  MoveL 686 to (-94.83, -177.34, 370.15) mm, rotated rx -20.04 ry 0.01 rz 0 deg; joints [12.615, -131.611, -68.908, -59.593, 88.727, 7.17]
  MoveL 687 to (-95.13, -172.76, 368.52) mm, rotated rx -19.93 ry 0.38 rz -0.14 deg; joints [12.853, -130.937, -70.265, -58.86, 88.278, 7.403]
  MoveL 688 to (-95.18, -165.44, 365.46) mm, rotated rx -20.3 ry 0.73 rz -0.27 deg; joints [13.07, -130.12, -71.703, -58.656, 87.921, 7.628]
  MoveL 689 to (-94.96, -155.27, 361.72) mm, rotated rx -19.76 ry 0.12 rz -0.04 deg; joints [12.925, -128.559, -74.952, -56.346, 88.521, 7.469]
  MoveL 690 to (-95.06, -148.96, 360) mm, rotated rx -19.41 ry -0.34 rz 0.12 deg; joints [12.816, -127.682, -76.899, -54.857, 88.972, 7.352]
  MoveL 691 to (-89.88, -148.96, 360) mm, rotated rx -19.07 ry -0.33 rz 0.11 deg; joints [12.421, -127.542, -77.28, -54.28, 88.998, 6.956]
  MoveL 692 to (-94.67, -143.58, 357.81) mm, rotated rx -19.21 ry -0.64 rz 0.22 deg; joints [12.719, -126.92, -78.436, -53.844, 89.284, 7.251]
  MoveL 693 to (-95.24, -134.75, 355.85) mm, rotated rx -19.89 ry -0.83 rz 0.3 deg; joints [12.73, -126.323, -79.629, -53.895, 89.571, 7.278]
  MoveL 694 to (-95.24, -124.99, 352.14) mm, rotated rx -20.45 ry -1.05 rz 0.39 deg; joints [12.704, -125.412, -81.243, -53.713, 89.885, 7.264]
  MoveL 695 to (-92.42, -119.21, 350) mm, rotated rx -20.35 ry -1.23 rz 0.46 deg; joints [12.457, -124.708, -82.656, -52.889, 90.101, 7.019]
  MoveL 696 to (-95.21, -114.33, 347.08) mm, rotated rx -20.45 ry -1.17 rz 0.44 deg; joints [12.774, -124.04, -83.727, -52.59, 89.995, 7.334]
  MoveL 697 to (-95.11, -104.56, 343.32) mm, rotated rx -20.25 ry -1.28 rz 0.47 deg; joints [12.838, -122.816, -86.139, -51.19, 90.078, 7.393]
  MoveL 698 to (-95.03, -94.94, 340.98) mm, rotated rx -19.38 ry -1.18 rz 0.41 deg; joints [13.046, -121.51, -89.146, -48.641, 89.811, 7.577]
  MoveL 699 to (-91.55, -89.14, 340) mm, rotated rx -19.07 ry -1.15 rz 0.4 deg; joints [12.839, -120.897, -90.647, -47.446, 89.781, 7.365]
  MoveL 700 to (-95.44, -84.4, 336.73) mm, rotated rx -19.11 ry -1.33 rz 0.46 deg; joints [13.163, -120.206, -91.7, -47.101, 89.907, 7.684]
  MoveL 701 to (-95.05, -75.22, 333) mm, rotated rx -20.06 ry -1.49 rz 0.54 deg; joints [13.102, -119.543, -92.613, -47.764, 90.223, 7.648]
  MoveL 702 to (-95.12, -66.84, 330.77) mm, rotated rx -20.48 ry -1.53 rz 0.57 deg; joints [13.159, -118.908, -93.858, -47.567, 90.322, 7.714]
  MoveL 703 to (-95.11, -61.19, 328.48) mm, rotated rx -20.08 ry -1.43 rz 0.52 deg; joints [13.317, -118.116, -95.454, -46.38, 90.126, 7.86]
  MoveL 704 to (-94.95, -54.68, 325.45) mm, rotated rx -20.03 ry -1.3 rz 0.47 deg; joints [13.468, -117.321, -96.854, -45.745, 89.952, 8.008]
  MoveL 705 to (-95.13, -44.85, 322.06) mm, rotated rx -19.59 ry -1.28 rz 0.45 deg; joints [13.666, -116.156, -99.258, -44.08, 89.831, 8.191]
  MoveL 706 to (-93.28, -38.74, 320) mm, rotated rx -19.37 ry -1.41 rz 0.49 deg; joints [13.524, -115.48, -100.669, -43.099, 89.961, 8.045]
  MoveL 707 to (-95.27, -34.68, 317.51) mm, rotated rx -19.05 ry -1.44 rz 0.5 deg; joints [13.789, -114.821, -101.831, -42.28, 89.901, 8.297]
  MoveL 708 to (-95, -25.83, 315.53) mm, rotated rx -19.14 ry -1.47 rz 0.51 deg; joints [13.868, -114.108, -103.402, -41.504, 89.923, 8.377]
  MoveL 709 to (-95.26, -15.36, 311.91) mm, rotated rx -18.64 ry -1.49 rz 0.5 deg; joints [14.085, -112.917, -105.883, -39.713, 89.831, 8.575]
  MoveL 710 to (-94.57, -9.01, 310) mm, rotated rx -18.16 ry -1.4 rz 0.46 deg; joints [14.208, -112.189, -107.516, -38.36, 89.638, 8.681]
  MoveL 711 to (-94.8, -3.67, 307.71) mm, rotated rx -17.94 ry -1.19 rz 0.39 deg; joints [14.466, -111.532, -108.75, -37.596, 89.329, 8.926]
  MoveL 712 to (-94.93, 5.41, 304.51) mm, rotated rx -17.3 ry -1.12 rz 0.35 deg; joints [14.744, -110.468, -111.026, -35.775, 89.086, 9.176]
  MoveL 713 to (-95.04, 14.85, 302.51) mm, rotated rx -17.21 ry -1.01 rz 0.31 deg; joints [14.992, -109.714, -112.788, -34.694, 88.907, 9.414]
  MoveL 714 to (-94.95, 23.14, 300.98) mm, rotated rx -17.62 ry -1.13 rz 0.36 deg; joints [15.02, -109.237, -113.848, -34.497, 89.087, 9.457]
  MoveL 715 to (-95.55, 28.29, 298.3) mm, rotated rx -18.2 ry -1.07 rz 0.35 deg; joints [15.17, -108.771, -114.269, -35.132, 89.097, 9.625]
  MoveL 716 to (-95.03, 35.17, 294.87) mm, rotated rx -19.11 ry -0.94 rz 0.33 deg; joints [15.247, -108.211, -114.702, -36.172, 89.104, 9.73]
  MoveL 717 to (-94.91, 45.46, 291.79) mm, rotated rx -19.49 ry -1.08 rz 0.38 deg; joints [15.308, -107.423, -116.156, -35.863, 89.307, 9.803]
  MoveL 718 to (-93.25, 51.3, 290) mm, rotated rx -18.82 ry -1.28 rz 0.44 deg; joints [15.184, -106.745, -117.783, -34.216, 89.42, 9.659]
  MoveL 719 to (-95.13, 55.87, 287.9) mm, rotated rx -18.18 ry -1.04 rz 0.34 deg; joints [15.727, -106.043, -119.212, -32.903, 88.951, 10.169]
  MoveL 720 to (-95.02, 65.32, 284.92) mm, rotated rx -17.88 ry -0.65 rz 0.21 deg; joints [16.219, -105.1, -121.129, -31.723, 88.389, 10.641]
  MoveL 721 to (-94.97, 75, 282.29) mm, rotated rx -17.01 ry -0.47 rz 0.14 deg; joints [16.669, -104.106, -123.55, -29.499, 87.945, 11.045]
  MoveL 722 to (-95.57, 81.71, 280.31) mm, rotated rx -16.74 ry -0.5 rz 0.15 deg; joints [16.933, -103.484, -124.933, -28.476, 87.854, 11.29]
  MoveL 723 to (-94.86, 86.85, 278.18) mm, rotated rx -16.68 ry -0.56 rz 0.17 deg; joints [16.947, -102.95, -125.872, -27.996, 87.91, 11.3]
  MoveL 724 to (-95.16, 94.95, 276.16) mm, rotated rx -16.91 ry -0.57 rz 0.17 deg; joints [17.159, -102.378, -127.022, -27.649, 87.916, 11.518]
  MoveL 725 to (-96.68, 102.58, 275.65) mm, rotated rx -15.92 ry -0.81 rz 0.23 deg; joints [17.522, -101.885, -129.109, -25.048, 87.866, 11.821]
  MoveL 726 to (-84.81, -254.16, 398.04) mm, rotated rx -18.14 ry -0.49 rz 0.16 deg; joints [11.089, -142.234, -48.176, -67.726, 89.323, 5.629]
  MoveL 727 to (-84.83, -246.42, 397.43) mm, rotated rx -19.51 ry -0.51 rz 0.18 deg; joints [11.08, -142.169, -48.262, -69.063, 89.483, 5.647]
  MoveL 728 to (-84.96, -235.69, 393.28) mm, rotated rx -20.66 ry -0.69 rz 0.26 deg; joints [11.053, -141.138, -50.022, -69.462, 89.799, 5.64]
  MoveL 729 to (-84.27, -228.62, 390.27) mm, rotated rx -20.97 ry -1.13 rz 0.43 deg; joints [10.868, -140.127, -51.941, -68.816, 90.332, 5.462]
  MoveL 730 to (-85.04, -223.33, 387.97) mm, rotated rx -21.99 ry -1.35 rz 0.55 deg; joints [10.834, -139.957, -52.001, -69.91, 90.674, 5.445]
  MoveL 731 to (-84.87, -214.7, 385.26) mm, rotated rx -22.47 ry -1.84 rz 0.76 deg; joints [10.661, -138.951, -54.007, -69.339, 91.279, 5.28]
  MoveL 732 to (-84.93, -206.09, 382.19) mm, rotated rx -22.25 ry -2.23 rz 0.91 deg; joints [10.573, -137.441, -57.118, -67.482, 91.687, 5.191]
  MoveL 733 to (-85.21, -200.4, 379) mm, rotated rx -21.97 ry -2.25 rz 0.91 deg; joints [10.642, -136.244, -59.41, -66.099, 91.667, 5.255]
  MoveL 734 to (-84.67, -194.51, 376.22) mm, rotated rx -21.82 ry -2.22 rz 0.89 deg; joints [10.665, -135.201, -61.427, -64.985, 91.616, 5.276]
  MoveL 735 to (-85.3, -184.88, 372.55) mm, rotated rx -21.44 ry -1.6 rz 0.63 deg; joints [11.069, -133.516, -64.805, -62.969, 90.844, 5.669]
  MoveL 736 to (-85.21, -177.44, 370.35) mm, rotated rx -20.98 ry -0.87 rz 0.33 deg; joints [11.454, -132.242, -67.486, -61.195, 89.957, 6.042]
  MoveL 737 to (-85.03, -172.64, 368.48) mm, rotated rx -20.75 ry -0.44 rz 0.17 deg; joints [11.679, -131.432, -69.11, -60.203, 89.44, 6.26]
  MoveL 738 to (-84.94, -165.44, 365.46) mm, rotated rx -20.37 ry -0.12 rz 0.04 deg; joints [11.9, -130.218, -71.536, -58.653, 89.017, 6.471]
  MoveL 739 to (-85.48, -155.44, 361.28) mm, rotated rx -19.25 ry -0.04 rz 0.01 deg; joints [12.13, -128.312, -75.522, -55.479, 88.766, 6.675]
  MoveL 740 to (-82.13, -150.42, 359) mm, rotated rx -18.73 ry -0.38 rz 0.13 deg; joints [11.782, -127.423, -77.38, -53.941, 89.136, 6.321]
  MoveL 741 to (-84.91, -144.97, 357.61) mm, rotated rx -18.63 ry -0.52 rz 0.18 deg; joints [12.002, -126.775, -78.786, -53.071, 89.225, 6.534]
  MoveL 742 to (-85.11, -135.15, 355.64) mm, rotated rx -19.31 ry -0.98 rz 0.34 deg; joints [11.863, -126.118, -80.166, -52.971, 89.812, 6.412]
  MoveL 743 to (-84.89, -125.22, 352.31) mm, rotated rx -20.49 ry -1.36 rz 0.51 deg; joints [11.702, -125.532, -81.043, -53.799, 90.384, 6.278]
  MoveL 744 to (-81.66, -120.69, 349) mm, rotated rx -21 ry -1.04 rz 0.4 deg; joints [11.61, -125.044, -81.552, -54.323, 90.118, 6.196]
  MoveL 745 to (-87.84, -119.21, 350) mm, rotated rx -20.58 ry -1.12 rz 0.42 deg; joints [12.117, -124.823, -82.364, -53.302, 90.066, 6.689]
  MoveL 746 to (-84.74, -114.13, 347.26) mm, rotated rx -20.77 ry -0.68 rz 0.26 deg; joints [12.109, -124.213, -83.322, -53.205, 89.633, 6.684]
  MoveL 747 to (-84.88, -104.45, 343.56) mm, rotated rx -19.91 ry -0.89 rz 0.32 deg; joints [12.172, -122.715, -86.477, -50.661, 89.737, 6.729]
  MoveL 748 to (-85.9, -95.32, 340.81) mm, rotated rx -19.48 ry -1.14 rz 0.4 deg; joints [12.262, -121.594, -88.906, -48.897, 89.928, 6.808]
  MoveL 749 to (-81.76, -91.98, 339) mm, rotated rx -19.35 ry -0.99 rz 0.35 deg; joints [12.018, -121.119, -89.755, -48.418, 89.804, 6.566]
  MoveL 750 to (-87.55, -89.14, 340) mm, rotated rx -19.04 ry -1.05 rz 0.36 deg; joints [12.537, -120.9, -90.648, -47.429, 89.732, 7.068]
  MoveL 751 to (-84.71, -84.61, 337.65) mm, rotated rx -18.99 ry -0.91 rz 0.31 deg; joints [12.417, -120.311, -91.674, -46.96, 89.595, 6.95]
  MoveL 752 to (-84.95, -75.08, 332.91) mm, rotated rx -19.86 ry -1.04 rz 0.37 deg; joints [12.44, -119.469, -92.789, -47.532, 89.836, 6.991]
  MoveL 753 to (-84.91, -66.88, 330.61) mm, rotated rx -20.34 ry -1.25 rz 0.46 deg; joints [12.388, -118.87, -93.932, -47.437, 90.136, 6.951]
  MoveL 754 to (-85.07, -61.26, 328.67) mm, rotated rx -20.11 ry -1.4 rz 0.51 deg; joints [12.408, -118.2, -95.324, -46.46, 90.256, 6.966]
  MoveL 755 to (-85.02, -54.81, 325.82) mm, rotated rx -20 ry -1.41 rz 0.51 deg; joints [12.487, -117.418, -96.765, -45.692, 90.238, 7.041]
  MoveL 756 to (-84.99, -44.93, 322.16) mm, rotated rx -19.53 ry -1.38 rz 0.49 deg; joints [12.653, -116.206, -99.224, -43.982, 90.116, 7.194]
  MoveL 757 to (-83.93, -37.55, 320.41) mm, rotated rx -19.24 ry -1.48 rz 0.52 deg; joints [12.61, -115.476, -100.91, -42.732, 90.187, 7.144]
  MoveL 758 to (-85.47, -33.08, 317.84) mm, rotated rx -19.11 ry -1.45 rz 0.5 deg; joints [12.846, -114.844, -101.966, -42.181, 90.096, 7.373]
  MoveL 759 to (-85.27, -25.33, 315.56) mm, rotated rx -19.07 ry -1.36 rz 0.47 deg; joints [12.978, -114.107, -103.479, -41.378, 89.976, 7.502]
  MoveL 760 to (-84.89, -15.77, 311.74) mm, rotated rx -18.78 ry -1.43 rz 0.49 deg; joints [13.062, -113.012, -105.595, -40.06, 89.988, 7.577]
  MoveL 761 to (-85.09, -9.98, 310) mm, rotated rx -18.54 ry -1.27 rz 0.42 deg; joints [13.276, -112.393, -106.913, -39.149, 89.74, 7.78]
  MoveL 762 to (-84.8, -4.2, 307.93) mm, rotated rx -18.18 ry -1.05 rz 0.35 deg; joints [13.484, -111.701, -108.347, -38.08, 89.423, 7.974]
  MoveL 763 to (-85.06, 5.28, 305.8) mm, rotated rx -17.23 ry -0.91 rz 0.28 deg; joints [13.814, -110.671, -110.953, -35.594, 89.068, 8.266]
  MoveL 764 to (-84.99, 14.63, 301.76) mm, rotated rx -17.22 ry -1.15 rz 0.36 deg; joints [13.828, -109.688, -112.682, -34.803, 89.309, 8.279]
  MoveL 765 to (-85.77, 22.24, 300.18) mm, rotated rx -17.6 ry -1.07 rz 0.34 deg; joints [14.047, -109.203, -113.681, -34.672, 89.237, 8.506]
  MoveL 766 to (-84.15, 26.99, 298.69) mm, rotated rx -18.27 ry -1 rz 0.33 deg; joints [13.935, -108.96, -113.894, -35.376, 89.288, 8.417]
  MoveL 767 to (-85.02, 35.35, 295.86) mm, rotated rx -18.92 ry -1.06 rz 0.36 deg; joints [14.081, -108.355, -114.793, -35.714, 89.42, 8.58]
  MoveL 768 to (-85, 45.69, 292.45) mm, rotated rx -19.11 ry -1.58 rz 0.55 deg; joints [13.917, -107.501, -116.427, -35.041, 90.025, 8.424]
  MoveL 769 to (-84.93, 51.88, 290) mm, rotated rx -18.91 ry -1.75 rz 0.6 deg; joints [13.931, -106.837, -117.708, -34.199, 90.171, 8.432]
  MoveL 770 to (-85.15, 56.65, 288) mm, rotated rx -18.6 ry -1.62 rz 0.55 deg; joints [14.16, -106.243, -118.85, -33.365, 89.943, 8.648]
  MoveL 771 to (-85.04, 65.47, 285.53) mm, rotated rx -18.18 ry -1.37 rz 0.45 deg; joints [14.519, -105.381, -120.759, -31.946, 89.541, 8.986]
  MoveL 772 to (-85.04, 75.21, 282.85) mm, rotated rx -17.29 ry -1.1 rz 0.34 deg; joints [14.99, -104.363, -123.22, -29.684, 89.016, 9.415]
  MoveL 773 to (-85.08, 80.94, 280) mm, rotated rx -16.76 ry -0.95 rz 0.29 deg; joints [15.294, -103.572, -124.713, -28.488, 88.702, 9.692]
  MoveL 774 to (-84.92, 86.24, 278.23) mm, rotated rx -16.55 ry -0.92 rz 0.27 deg; joints [15.443, -103.052, -125.802, -27.719, 88.597, 9.828]
  MoveL 775 to (-84.97, 94.98, 276.23) mm, rotated rx -16.7 ry -0.91 rz 0.27 deg; joints [15.634, -102.45, -127.114, -27.169, 88.572, 10.021]
  MoveL 776 to (-85.97, 101.04, 275.32) mm, rotated rx -15.86 ry -0.92 rz 0.26 deg; joints [16.001, -101.951, -128.843, -25.117, 88.344, 10.341]
  MoveL 777 to (-73.01, -256.67, 400.33) mm, rotated rx -16.93 ry -1.96 rz 0.6 deg; joints [9.707, -142.108, -49.069, -65.622, 91.046, 4.257]
  MoveL 778 to (-76.07, -253.64, 398.85) mm, rotated rx -17.91 ry -1.49 rz 0.48 deg; joints [10.094, -142.199, -48.515, -67.094, 90.552, 4.652]
  MoveL 779 to (-74.72, -245.59, 396.62) mm, rotated rx -19.49 ry -1.5 rz 0.53 deg; joints [9.986, -142.077, -48.436, -68.867, 90.733, 4.572]
  MoveL 780 to (-75.3, -235.91, 394.03) mm, rotated rx -20.25 ry -1.47 rz 0.54 deg; joints [10.071, -141.051, -50.447, -68.643, 90.751, 4.666]
  MoveL 781 to (-74.37, -228.01, 391.14) mm, rotated rx -20.89 ry -1.46 rz 0.56 deg; joints [10.035, -140.182, -52.039, -68.557, 90.806, 4.64]
  MoveL 782 to (-75.54, -222.35, 388.11) mm, rotated rx -21.63 ry -1.6 rz 0.64 deg; joints [10.073, -139.664, -52.77, -69.061, 91.019, 4.687]
  MoveL 783 to (-74.76, -215.31, 386) mm, rotated rx -21.85 ry -2.02 rz 0.81 deg; joints [9.881, -138.752, -54.644, -68.29, 91.514, 4.5]
  MoveL 784 to (-75.09, -205.73, 383.37) mm, rotated rx -22.06 ry -2.43 rz 0.98 deg; joints [9.784, -137.492, -57.28, -67.082, 91.984, 4.408]
  MoveL 785 to (-72.03, -198.94, 380) mm, rotated rx -21.9 ry -2.35 rz 0.94 deg; joints [9.641, -136.268, -59.63, -65.813, 91.907, 4.264]
  MoveL 786 to (-75.36, -193.98, 376.92) mm, rotated rx -21.93 ry -2.43 rz 0.98 deg; joints [9.883, -135.377, -61.211, -65.133, 91.965, 4.504]
  MoveL 787 to (-75.05, -184.85, 373.44) mm, rotated rx -22.22 ry -2.31 rz 0.94 deg; joints [9.958, -134.205, -63.446, -64.361, 91.853, 4.581]
  MoveL 788 to (-74.7, -177.25, 370.46) mm, rotated rx -21.92 ry -1.94 rz 0.78 deg; joints [10.155, -132.91, -66.031, -62.811, 91.393, 4.772]
  MoveL 789 to (-75.37, -172.64, 368.47) mm, rotated rx -21.36 ry -1.69 rz 0.66 deg; joints [10.367, -131.901, -68.107, -61.211, 91.045, 4.974]
  MoveL 790 to (-75.25, -165.22, 365.42) mm, rotated rx -20.52 ry -1.5 rz 0.56 deg; joints [10.531, -130.404, -71.223, -58.774, 90.732, 5.123]
  MoveL 791 to (-74.56, -155.22, 361.43) mm, rotated rx -19.46 ry -1.21 rz 0.43 deg; joints [10.726, -128.537, -75.133, -55.707, 90.287, 5.298]
  MoveL 792 to (-77.9, -150.42, 359) mm, rotated rx -18.71 ry -0.69 rz 0.23 deg; joints [11.306, -127.452, -77.352, -53.877, 89.546, 5.853]
  MoveL 793 to (-72.07, -146.71, 360.32) mm, rotated rx -18.67 ry -1 rz 0.34 deg; joints [10.716, -127.347, -78.044, -53.219, 89.984, 5.274]
  MoveL 794 to (-76.15, -143.92, 358.03) mm, rotated rx -18.55 ry -0.76 rz 0.26 deg; joints [11.19, -126.767, -78.99, -52.758, 89.628, 5.736]
  MoveL 795 to (-75.08, -135.23, 355.09) mm, rotated rx -18.82 ry -0.87 rz 0.3 deg; joints [11.114, -125.893, -80.672, -52.208, 89.786, 5.667]
  MoveL 796 to (-74.48, -125.62, 351.28) mm, rotated rx -20.43 ry -1.36 rz 0.51 deg; joints [10.848, -125.484, -80.965, -53.873, 90.518, 5.435]
  MoveL 797 to (-76.64, -120.69, 349) mm, rotated rx -21.19 ry -1.33 rz 0.51 deg; joints [11.051, -125.183, -81.253, -54.645, 90.532, 5.647]
  MoveL 798 to (-74.95, -114.72, 347.47) mm, rotated rx -21.07 ry -1.3 rz 0.5 deg; joints [10.978, -124.511, -82.71, -53.744, 90.499, 5.573]
  MoveL 799 to (-75.1, -104.46, 343.25) mm, rotated rx -19.75 ry -1.05 rz 0.38 deg; joints [11.268, -122.681, -86.561, -50.434, 90.047, 5.836]
  MoveL 800 to (-75.85, -97.4, 340.22) mm, rotated rx -19.53 ry -0.91 rz 0.32 deg; joints [11.48, -121.733, -88.379, -49.362, 89.84, 6.04]
  MoveL 801 to (-74.53, -92.78, 338.89) mm, rotated rx -19.56 ry -0.88 rz 0.31 deg; joints [11.423, -121.281, -89.311, -48.913, 89.818, 5.985]
  MoveL 802 to (-74.96, -84.95, 337.7) mm, rotated rx -19.29 ry -0.66 rz 0.23 deg; joints [11.654, -120.497, -91.203, -47.563, 89.514, 6.207]
  MoveL 803 to (-75.02, -75.28, 333.65) mm, rotated rx -19.56 ry -0.68 rz 0.24 deg; joints [11.74, -119.494, -92.957, -47.082, 89.547, 6.296]
  MoveL 804 to (-75.03, -66.77, 330.78) mm, rotated rx -20.12 ry -0.86 rz 0.32 deg; joints [11.706, -118.835, -94.101, -47.13, 89.81, 6.274]
  MoveL 805 to (-74.93, -61.27, 328.52) mm, rotated rx -20.15 ry -0.84 rz 0.31 deg; joints [11.767, -118.228, -95.207, -46.662, 89.78, 6.335]
  MoveL 806 to (-75.04, -54.83, 325.81) mm, rotated rx -20.09 ry -0.89 rz 0.33 deg; joints [11.824, -117.484, -96.585, -45.966, 89.82, 6.39]
  MoveL 807 to (-74.95, -44.87, 322.69) mm, rotated rx -19.29 ry -1.13 rz 0.39 deg; joints [11.849, -116.235, -99.358, -43.618, 89.969, 6.398]
  MoveL 808 to (-74.96, -37.09, 320.66) mm, rotated rx -19.06 ry -1.38 rz 0.48 deg; joints [11.811, -115.477, -101.065, -42.413, 90.217, 6.356]
  MoveL 809 to (-74.96, -31.8, 317.97) mm, rotated rx -19.05 ry -1.58 rz 0.54 deg; joints [11.77, -114.853, -102.124, -41.945, 90.429, 6.316]
  MoveL 810 to (-74.99, -24.39, 315.9) mm, rotated rx -19 ry -1.68 rz 0.58 deg; joints [11.801, -114.173, -103.57, -41.115, 90.528, 6.345]
  MoveL 811 to (-75.18, -15.17, 312.05) mm, rotated rx -18.74 ry -1.72 rz 0.58 deg; joints [11.93, -113.101, -105.6, -39.892, 90.509, 6.466]
  MoveL 812 to (-74.06, -8.79, 310) mm, rotated rx -18.95 ry -1.65 rz 0.57 deg; joints [11.917, -112.568, -106.582, -39.655, 90.466, 6.458]
  MoveL 813 to (-75.47, -3.56, 308.41) mm, rotated rx -18.65 ry -1.41 rz 0.48 deg; joints [12.286, -111.965, -107.873, -38.698, 90.102, 6.812]
  MoveL 814 to (-74.83, 5.34, 306.12) mm, rotated rx -17.53 ry -0.9 rz 0.28 deg; joints [12.71, -110.865, -110.56, -36.079, 89.341, 7.199]
  MoveL 815 to (-74.98, 14.73, 301.9) mm, rotated rx -16.85 ry -0.95 rz 0.29 deg; joints [12.893, -109.665, -112.947, -34.205, 89.261, 7.356]
  MoveL 816 to (-73.78, 22.12, 300.05) mm, rotated rx -17.84 ry -0.93 rz 0.3 deg; joints [12.806, -109.332, -113.32, -35.15, 89.386, 7.3]
  MoveL 817 to (-75.84, 26.68, 298.86) mm, rotated rx -18.32 ry -0.88 rz 0.29 deg; joints [13.09, -109.066, -113.699, -35.531, 89.34, 7.592]
  MoveL 818 to (-75.01, 35.38, 296.67) mm, rotated rx -18.56 ry -0.99 rz 0.33 deg; joints [13.035, -108.443, -114.99, -35.08, 89.506, 7.544]
  MoveL 819 to (-74.93, 45.61, 292.44) mm, rotated rx -18.76 ry -1.17 rz 0.4 deg; joints [13.067, -107.453, -116.641, -34.59, 89.71, 7.581]
  MoveL 820 to (-74.95, 52.6, 290.22) mm, rotated rx -18.76 ry -1.25 rz 0.42 deg; joints [13.129, -106.834, -117.866, -33.97, 89.783, 7.641]
  MoveL 821 to (-75.19, 57.45, 288.1) mm, rotated rx -18.7 ry -1.33 rz 0.45 deg; joints [13.195, -106.306, -118.782, -33.515, 89.843, 7.705]
  MoveL 822 to (-74.95, 65.38, 285.7) mm, rotated rx -18.2 ry -1.36 rz 0.45 deg; joints [13.325, -105.5, -120.601, -32.002, 89.777, 7.818]
  MoveL 823 to (-75.05, 75.16, 282.86) mm, rotated rx -17.59 ry -1.52 rz 0.48 deg; joints [13.454, -104.559, -122.809, -30.105, 89.83, 7.925]
  MoveL 824 to (-74.24, 81.93, 280.2) mm, rotated rx -17.23 ry -1.36 rz 0.42 deg; joints [13.624, -103.803, -124.301, -29.037, 89.576, 8.08]
  MoveL 825 to (-75.48, 86.98, 278.59) mm, rotated rx -16.82 ry -1.12 rz 0.34 deg; joints [14.086, -103.244, -125.549, -27.987, 89.163, 8.517]
  MoveL 826 to (-74.63, 94.41, 277.05) mm, rotated rx -16.76 ry -1.01 rz 0.31 deg; joints [14.204, -102.723, -126.824, -27.193, 89.012, 8.631]
  MoveL 827 to (-65.15, -255.36, 401) mm, rotated rx -17.39 ry -2.76 rz 0.86 deg; joints [8.834, -142.503, -48.365, -66.343, 92.11, 3.415]
  MoveL 828 to (-68.33, -250.6, 399) mm, rotated rx -18.23 ry -2.26 rz 0.75 deg; joints [9.25, -142.185, -48.692, -67.201, 91.57, 3.832]
  MoveL 829 to (-61.71, -249.14, 400) mm, rotated rx -18.67 ry -2.75 rz 0.93 deg; joints [8.585, -142.564, -48.07, -67.864, 92.249, 3.187]
  MoveL 830 to (-65.42, -244.25, 397.74) mm, rotated rx -19.57 ry -2.44 rz 0.87 deg; joints [8.966, -142.253, -48.363, -68.786, 91.915, 3.571]
  MoveL 831 to (-64.63, -234.94, 394.33) mm, rotated rx -20.49 ry -2.11 rz 0.79 deg; joints [9.056, -141.293, -50.049, -68.996, 91.627, 3.669]
  MoveL 832 to (-65.83, -226.85, 390.87) mm, rotated rx -21.13 ry -1.58 rz 0.61 deg; joints [9.377, -140.272, -51.842, -68.9, 91.061, 3.992]
  MoveL 833 to (-65.03, -221.73, 388.6) mm, rotated rx -21.32 ry -1.61 rz 0.63 deg; joints [9.332, -139.518, -53.255, -68.431, 91.109, 3.95]
  MoveL 834 to (-64.86, -215.23, 385.75) mm, rotated rx -21.4 ry -1.63 rz 0.64 deg; joints [9.345, -138.462, -55.287, -67.535, 91.133, 3.964]
  MoveL 835 to (-65.13, -205.62, 383.18) mm, rotated rx -21.77 ry -1.76 rz 0.7 deg; joints [9.347, -137.311, -57.655, -66.674, 91.303, 3.971]
  MoveL 836 to (-64.72, -199.36, 380.8) mm, rotated rx -21.82 ry -1.88 rz 0.75 deg; joints [9.298, -136.391, -59.477, -65.815, 91.447, 3.923]
  MoveL 837 to (-65.23, -193.95, 378) mm, rotated rx -21.77 ry -2.06 rz 0.82 deg; joints [9.295, -135.46, -61.236, -64.914, 91.632, 3.919]
  MoveL 838 to (-65.1, -184.95, 373.73) mm, rotated rx -22.13 ry -2.52 rz 1.03 deg; joints [9.125, -134.306, -63.334, -64.297, 92.188, 3.756]
  MoveL 839 to (-64.74, -176.51, 370.94) mm, rotated rx -21.88 ry -2.91 rz 1.17 deg; joints [8.983, -133.032, -66.004, -62.624, 92.601, 3.614]
  MoveL 840 to (-65.61, -171.78, 369) mm, rotated rx -21.31 ry -2.89 rz 1.13 deg; joints [9.103, -132.024, -68.109, -60.961, 92.512, 3.727]
  MoveL 841 to (-65.18, -165.73, 366) mm, rotated rx -20.82 ry -2.85 rz 1.08 deg; joints [9.14, -130.857, -70.424, -59.32, 92.42, 3.757]
  MoveL 842 to (-64.97, -155.25, 361.25) mm, rotated rx -20.11 ry -2.4 rz 0.88 deg; joints [9.408, -129.005, -74.09, -56.834, 91.84, 4.013]
  MoveL 843 to (-65.75, -146.4, 360.31) mm, rotated rx -19.19 ry -1.57 rz 0.54 deg; joints [9.929, -127.651, -77.351, -54.073, 90.782, 4.511]
  MoveL 844 to (-63.43, -142.11, 358.75) mm, rotated rx -18.97 ry -1.54 rz 0.53 deg; joints [9.79, -127.05, -78.607, -53.203, 90.763, 4.371]
  MoveL 845 to (-64.91, -135.19, 355.93) mm, rotated rx -18.49 ry -1.26 rz 0.42 deg; joints [10.105, -125.946, -80.865, -51.592, 90.368, 4.672]
  MoveL 846 to (-64.96, -125.47, 351.95) mm, rotated rx -19.97 ry -1.58 rz 0.57 deg; joints [9.977, -125.432, -81.36, -53.06, 90.854, 4.569]
  MoveL 847 to (-65.15, -115.05, 348.49) mm, rotated rx -21.29 ry -2.02 rz 0.79 deg; joints [9.804, -124.882, -82.15, -54.09, 91.471, 4.417]
  MoveL 848 to (-64.82, -104.77, 343.35) mm, rotated rx -20.2 ry -1.8 rz 0.66 deg; joints [10.001, -123.043, -85.791, -51.226, 91.111, 4.597]
  MoveL 849 to (-64.52, -97.49, 340.2) mm, rotated rx -19.78 ry -1.47 rz 0.53 deg; joints [10.21, -121.97, -87.892, -49.811, 90.683, 4.796]
  MoveL 850 to (-65.76, -92.61, 338.71) mm, rotated rx -19.75 ry -1.15 rz 0.41 deg; joints [10.517, -121.412, -89.011, -49.245, 90.283, 5.097]
  MoveL 851 to (-64.85, -84.95, 337.44) mm, rotated rx -19.58 ry -1.04 rz 0.37 deg; joints [10.555, -120.685, -90.743, -48.084, 90.146, 5.132]
  MoveL 852 to (-65.11, -75.24, 333.77) mm, rotated rx -19.53 ry -0.8 rz 0.29 deg; joints [10.785, -119.58, -92.857, -47.047, 89.85, 5.357]
  MoveL 853 to (-65.17, -67.71, 331) mm, rotated rx -20.06 ry -0.74 rz 0.27 deg; joints [10.864, -118.968, -93.855, -47.197, 89.826, 5.444]
  MoveL 854 to (-64.88, -61.99, 328.54) mm, rotated rx -20.08 ry -0.81 rz 0.29 deg; joints [10.859, -118.327, -95.016, -46.686, 89.895, 5.439]
  MoveL 855 to (-64.91, -54.78, 325.83) mm, rotated rx -19.78 ry -0.92 rz 0.33 deg; joints [10.888, -117.452, -96.784, -45.486, 89.976, 5.463]
  MoveL 856 to (-65, -45, 322.9) mm, rotated rx -18.97 ry -1.19 rz 0.41 deg; joints [10.883, -116.249, -99.508, -43.134, 90.186, 5.443]
  MoveL 857 to (-65.11, -36.96, 320.68) mm, rotated rx -18.76 ry -1.49 rz 0.51 deg; joints [10.82, -115.465, -101.247, -41.934, 90.488, 5.377]
  MoveL 858 to (-64.74, -31.76, 318.06) mm, rotated rx -18.76 ry -1.66 rz 0.56 deg; joints [10.744, -114.862, -102.27, -41.496, 90.683, 5.303]
  MoveL 859 to (-64.97, -24.3, 315.95) mm, rotated rx -18.97 ry -1.76 rz 0.61 deg; joints [10.77, -114.261, -103.467, -41.099, 90.806, 5.333]
  MoveL 860 to (-65.08, -14.99, 312.31) mm, rotated rx -18.83 ry -1.66 rz 0.57 deg; joints [10.941, -113.24, -105.397, -40.058, 90.65, 5.497]
  MoveL 861 to (-66.46, -9.98, 310) mm, rotated rx -18.83 ry -1.66 rz 0.57 deg; joints [11.134, -112.662, -106.384, -39.645, 90.616, 5.687]
  MoveL 862 to (-65.01, -4.92, 308.34) mm, rotated rx -18.82 ry -1.81 rz 0.62 deg; joints [10.954, -112.21, -107.297, -39.164, 90.809, 5.511]
  MoveL 863 to (-64.9, 5.39, 306.11) mm, rotated rx -18.03 ry -1.63 rz 0.53 deg; joints [11.203, -111.153, -109.915, -36.834, 90.476, 5.738]
  MoveL 864 to (-64.99, 14.8, 302.51) mm, rotated rx -17.17 ry -0.86 rz 0.27 deg; joints [11.837, -109.914, -112.509, -34.713, 89.445, 6.337]
  MoveL 865 to (-65.2, 21.19, 300.38) mm, rotated rx -17.83 ry -0.49 rz 0.16 deg; joints [12.12, -109.461, -113.073, -35.309, 89.079, 6.63]
  MoveL 866 to (-64.85, 26.51, 298.5) mm, rotated rx -18.2 ry -0.47 rz 0.16 deg; joints [12.142, -109.055, -113.68, -35.482, 89.096, 6.661]
  MoveL 867 to (-65.27, 35.43, 297.32) mm, rotated rx -18.45 ry -0.61 rz 0.2 deg; joints [12.198, -108.562, -114.971, -34.915, 89.253, 6.722]
  MoveL 868 to (-65.11, 45.49, 292.37) mm, rotated rx -18.76 ry -0.77 rz 0.26 deg; joints [12.209, -107.506, -116.512, -34.718, 89.457, 6.74]
  MoveL 869 to (-64.38, 53.3, 290.45) mm, rotated rx -18.68 ry -0.73 rz 0.25 deg; joints [12.261, -106.874, -117.928, -33.855, 89.399, 6.789]
  MoveL 870 to (-65.66, 58.05, 288.62) mm, rotated rx -18.46 ry -0.88 rz 0.29 deg; joints [12.4, -106.349, -118.978, -33.092, 89.502, 6.919]
  MoveL 871 to (-65.1, 65.51, 285.99) mm, rotated rx -17.93 ry -1.1 rz 0.36 deg; joints [12.344, -105.554, -120.725, -31.589, 89.677, 6.851]
  MoveL 872 to (-64.95, 75.28, 282.96) mm, rotated rx -17.6 ry -1.11 rz 0.35 deg; joints [12.494, -104.639, -122.693, -30.205, 89.616, 6.989]
  MoveL 873 to (-64.8, 83.02, 280.36) mm, rotated rx -17.42 ry -1.09 rz 0.34 deg; joints [12.63, -103.905, -124.174, -29.283, 89.542, 7.117]
  MoveL 874 to (-65.73, 87.99, 278.81) mm, rotated rx -17.39 ry -1.24 rz 0.39 deg; joints [12.73, -103.478, -125.04, -28.8, 89.668, 7.214]
  MoveL 875 to (-64.91, 94.9, 276.86) mm, rotated rx -16.91 ry -1.49 rz 0.45 deg; joints [12.608, -102.873, -126.582, -27.353, 89.889, 7.08]
  MoveL 876 to (-63.79, 100.46, 275.17) mm, rotated rx -14.77 ry -1.97 rz 0.52 deg; joints [12.397, -102.17, -129.298, -23.151, 90.165, 6.81]
  MoveL 877 to (-55.08, -255.13, 401.19) mm, rotated rx -18.02 ry -3.09 rz 1.01 deg; joints [7.981, -143.156, -46.94, -67.751, 92.691, 2.589]
  MoveL 878 to (-56.48, -249.14, 400) mm, rotated rx -18.73 ry -2.93 rz 0.99 deg; joints [8.146, -142.695, -47.81, -68.05, 92.531, 2.757]
  MoveL 879 to (-55.08, -243.89, 398.03) mm, rotated rx -19.6 ry -2.86 rz 1.02 deg; joints [8.073, -142.439, -48.085, -68.909, 92.527, 2.693]
  MoveL 880 to (-55.32, -234.78, 394.56) mm, rotated rx -21.46 ry -2.55 rz 1 deg; joints [8.2, -142.235, -47.997, -71.075, 92.297, 2.834]
  MoveL 881 to (-54.6, -226.52, 391.17) mm, rotated rx -21.82 ry -1.82 rz 0.73 deg; joints [8.463, -140.953, -50.398, -70.357, 91.507, 3.096]
  MoveL 882 to (-55.44, -221.96, 389) mm, rotated rx -21.73 ry -1.37 rz 0.54 deg; joints [8.731, -139.989, -52.261, -69.389, 90.971, 3.359]
  MoveL 883 to (-55.07, -214.47, 384.68) mm, rotated rx -21.54 ry -0.94 rz 0.37 deg; joints [8.923, -138.406, -55.228, -67.848, 90.469, 3.547]
  MoveL 884 to (-54.94, -205, 382.03) mm, rotated rx -21.61 ry -1.01 rz 0.4 deg; joints [8.924, -137.061, -58.03, -66.458, 90.553, 3.549]
  MoveL 885 to (-53.88, -198.61, 380.23) mm, rotated rx -21.22 ry -1.27 rz 0.49 deg; joints [8.777, -135.928, -60.49, -64.722, 90.828, 3.4]
  MoveL 886 to (-55.44, -193.81, 378) mm, rotated rx -21.09 ry -1.75 rz 0.68 deg; joints [8.716, -135.107, -62.112, -63.759, 91.343, 3.34]
  MoveL 887 to (-55.01, -184.94, 373.95) mm, rotated rx -21.23 ry -2.67 rz 1.04 deg; joints [8.331, -133.912, -64.399, -62.751, 92.396, 2.962]
  MoveL 888 to (-55.05, -175.73, 370.93) mm, rotated rx -21.66 ry -3.27 rz 1.3 deg; joints [8.101, -132.972, -66.265, -62.219, 93.103, 2.739]
  MoveL 889 to (-54.65, -170.04, 369) mm, rotated rx -21.31 ry -3.28 rz 1.28 deg; joints [8.099, -132.022, -68.264, -60.823, 93.086, 2.734]
  MoveL 890 to (-54.85, -164.41, 366.05) mm, rotated rx -20.96 ry -3.1 rz 1.19 deg; joints [8.226, -130.96, -70.305, -59.498, 92.851, 2.857]
  MoveL 891 to (-55.49, -154.91, 362.11) mm, rotated rx -20.57 ry -2.93 rz 1.1 deg; joints [8.403, -129.452, -73.302, -57.624, 92.615, 3.028]
  MoveL 892 to (-54.08, -148.28, 360.39) mm, rotated rx -20.35 ry -2.66 rz 0.99 deg; joints [8.447, -128.583, -75.174, -56.423, 92.305, 3.069]
  MoveL 893 to (-55.48, -143.2, 358.42) mm, rotated rx -19.46 ry -2.33 rz 0.82 deg; joints [8.763, -127.47, -77.58, -54.254, 91.83, 3.37]
  MoveL 894 to (-55, -134.99, 356.02) mm, rotated rx -18.66 ry -1.84 rz 0.62 deg; joints [9.017, -126.162, -80.471, -51.913, 91.203, 3.609]
  MoveL 895 to (-54.98, -125.35, 352.2) mm, rotated rx -19.77 ry -1.45 rz 0.52 deg; joints [9.213, -125.455, -81.437, -52.786, 90.844, 3.815]
  MoveL 896 to (-51.67, -117.74, 350.23) mm, rotated rx -20.45 ry -1.66 rz 0.62 deg; joints [8.862, -125.015, -82.26, -53.068, 91.169, 3.477]
  MoveL 897 to (-55.97, -114.54, 348.45) mm, rotated rx -20.87 ry -1.89 rz 0.72 deg; joints [9.116, -124.734, -82.59, -53.413, 91.408, 3.732]
  MoveL 898 to (-55.09, -105.03, 345.47) mm, rotated rx -20.56 ry -2.05 rz 0.77 deg; joints [9.031, -123.584, -85.025, -51.812, 91.567, 3.645]
  MoveL 899 to (-54.78, -95.8, 341.3) mm, rotated rx -20.07 ry -1.97 rz 0.72 deg; joints [9.117, -122.238, -87.651, -50.04, 91.427, 3.725]
  MoveL 900 to (-55.59, -90.9, 339) mm, rotated rx -19.95 ry -1.89 rz 0.68 deg; joints [9.263, -121.572, -88.881, -49.364, 91.306, 3.867]
  MoveL 901 to (-55.11, -84.9, 337.25) mm, rotated rx -19.67 ry -1.91 rz 0.68 deg; joints [9.256, -120.861, -90.433, -48.239, 91.312, 3.857]
  MoveL 902 to (-55.03, -75.37, 334.07) mm, rotated rx -19.8 ry -1.91 rz 0.69 deg; joints [9.307, -119.914, -92.279, -47.467, 91.308, 3.908]
  MoveL 903 to (-54.87, -66.23, 331.06) mm, rotated rx -20.3 ry -1.64 rz 0.61 deg; joints [9.467, -119.148, -93.633, -47.405, 91.04, 4.072]
  MoveL 904 to (-55.99, -60.96, 328.81) mm, rotated rx -20.11 ry -1.35 rz 0.5 deg; joints [9.765, -118.438, -94.978, -46.597, 90.668, 4.362]
  MoveL 905 to (-54.91, -54.85, 326.1) mm, rotated rx -19.54 ry -1.42 rz 0.5 deg; joints [9.7, -117.543, -96.803, -45.093, 90.703, 4.291]
  MoveL 906 to (-54.88, -45, 322.49) mm, rotated rx -18.82 ry -1.52 rz 0.52 deg; joints [9.748, -116.278, -99.486, -42.949, 90.742, 4.327]
  MoveL 907 to (-55.06, -37.33, 320.37) mm, rotated rx -18.48 ry -1.49 rz 0.5 deg; joints [9.859, -115.46, -101.306, -41.609, 90.652, 4.431]
  MoveL 908 to (-55.03, -32.31, 318.59) mm, rotated rx -18.5 ry -1.64 rz 0.55 deg; joints [9.811, -114.981, -102.234, -41.175, 90.825, 4.384]
  MoveL 909 to (-55.04, -24.26, 316.54) mm, rotated rx -18.8 ry -1.87 rz 0.64 deg; joints [9.736, -114.399, -103.435, -40.827, 91.102, 4.315]
  MoveL 910 to (-54.89, -14.24, 312.77) mm, rotated rx -19.01 ry -2.06 rz 0.71 deg; joints [9.682, -113.469, -105.118, -40.268, 91.339, 4.266]
  MoveL 911 to (-54.05, -7.5, 310.39) mm, rotated rx -19.07 ry -1.71 rz 0.59 deg; joints [9.85, -112.802, -106.347, -39.792, 90.939, 4.431]
  MoveL 912 to (-55.83, -2.93, 308.4) mm, rotated rx -18.91 ry -1.48 rz 0.51 deg; joints [10.21, -112.216, -107.414, -39.177, 90.617, 4.782]
  MoveL 913 to (-54.99, 5.24, 305.93) mm, rotated rx -18.67 ry -1.34 rz 0.45 deg; joints [10.293, -111.403, -109.144, -38.028, 90.427, 4.859]
  MoveL 914 to (-54.93, 14.82, 302.64) mm, rotated rx -17.86 ry -0.72 rz 0.23 deg; joints [10.793, -110.21, -111.711, -35.908, 89.599, 5.333]
  MoveL 915 to (-54.36, 23.5, 300.49) mm, rotated rx -18.22 ry -0.41 rz 0.14 deg; joints [10.989, -109.587, -112.929, -35.705, 89.268, 5.533]
  MoveL 916 to (-56.75, 27.7, 298.7) mm, rotated rx -18.23 ry -0.25 rz 0.08 deg; joints [11.396, -109.106, -113.737, -35.415, 89.022, 5.932]
  MoveL 917 to (-54.99, 35.35, 296.21) mm, rotated rx -18.12 ry -0.47 rz 0.15 deg; joints [11.164, -108.422, -115.151, -34.548, 89.285, 5.702]
  MoveL 918 to (-54.77, 45.25, 292.41) mm, rotated rx -18.72 ry -0.68 rz 0.23 deg; joints [11.094, -107.622, -116.346, -34.727, 89.576, 5.646]
  MoveL 919 to (-56.11, 52.52, 290.89) mm, rotated rx -18.62 ry -0.69 rz 0.23 deg; joints [11.325, -107.049, -117.707, -33.837, 89.537, 5.871]
  MoveL 920 to (-54.38, 57.63, 288.36) mm, rotated rx -18.25 ry -0.72 rz 0.24 deg; joints [11.196, -106.396, -118.927, -32.898, 89.557, 5.736]
  MoveL 921 to (-55.11, 65.61, 285.92) mm, rotated rx -17.74 ry -0.86 rz 0.27 deg; joints [11.328, -105.594, -120.759, -31.351, 89.617, 5.854]
  MoveL 922 to (-55.08, 75.07, 283.06) mm, rotated rx -17.74 ry -0.95 rz 0.3 deg; joints [11.388, -104.8, -122.371, -30.516, 89.696, 5.912]
  MoveL 923 to (-54.96, 83.42, 280.64) mm, rotated rx -17.38 ry -1.03 rz 0.32 deg; joints [11.456, -104.052, -124.084, -29.195, 89.725, 5.97]
  MoveL 924 to (-55.01, 88.62, 278.67) mm, rotated rx -17.06 ry -1.07 rz 0.33 deg; joints [11.531, -103.494, -125.252, -28.262, 89.716, 6.036]
  MoveL 925 to (-55.4, 94.72, 276.82) mm, rotated rx -16.65 ry -1.08 rz 0.32 deg; joints [11.688, -102.908, -126.643, -27.046, 89.65, 6.179]
  MoveL 926 to (-59.53, 100.76, 276) mm, rotated rx -14.53 ry -1.76 rz 0.46 deg; joints [12.004, -102.311, -129.454, -22.648, 90.017, 6.424]
  MoveL 927 to (-46.34, -254.42, 400.9) mm, rotated rx -18.09 ry -2.41 rz 0.79 deg; joints [7.637, -143.145, -46.907, -67.918, 92.048, 2.252]
  MoveL 928 to (-41.13, -248.43, 400.2) mm, rotated rx -18.89 ry -2.07 rz 0.71 deg; joints [7.405, -142.908, -47.372, -68.515, 91.777, 2.03]
  MoveL 929 to (-45.49, -244.66, 398.21) mm, rotated rx -19.65 ry -2.43 rz 0.87 deg; joints [7.564, -142.715, -47.485, -69.328, 92.171, 2.192]
  MoveL 930 to (-44.87, -234.73, 394.47) mm, rotated rx -21.93 ry -2.36 rz 0.95 deg; joints [7.53, -142.75, -46.845, -72.211, 92.228, 2.174]
  MoveL 931 to (-45.1, -226.44, 391.15) mm, rotated rx -22.73 ry -1.99 rz 0.83 deg; joints [7.703, -141.823, -48.473, -72.324, 91.85, 2.349]
  MoveL 932 to (-46.29, -221.96, 389) mm, rotated rx -22.47 ry -1.59 rz 0.66 deg; joints [7.969, -140.709, -50.672, -71.002, 91.369, 2.611]
  MoveL 933 to (-45.31, -215.17, 386.08) mm, rotated rx -22.01 ry -1.24 rz 0.5 deg; joints [8.079, -139.139, -53.852, -68.945, 90.946, 2.716]
  MoveL 934 to (-45.07, -205.52, 383) mm, rotated rx -21.28 ry -1.15 rz 0.45 deg; joints [8.151, -137.14, -58.099, -65.973, 90.792, 2.783]
  MoveL 935 to (-44.78, -198.21, 380.5) mm, rotated rx -20.49 ry -1.53 rz 0.57 deg; joints [8.014, -135.593, -61.442, -63.371, 91.178, 2.641]
  MoveL 936 to (-44.78, -193.08, 378.33) mm, rotated rx -20.06 ry -1.92 rz 0.7 deg; joints [7.879, -134.596, -63.525, -61.841, 91.591, 2.505]
  MoveL 937 to (-45.1, -185.52, 374.93) mm, rotated rx -20.23 ry -2.65 rz 0.98 deg; joints [7.615, -133.621, -65.376, -61.098, 92.425, 2.247]
  MoveL 938 to (-45.08, -174.98, 371.44) mm, rotated rx -21.17 ry -3.38 rz 1.31 deg; joints [7.307, -132.825, -66.831, -61.35, 93.312, 1.95]
  MoveL 939 to (-41.71, -168.14, 370.29) mm, rotated rx -21.32 ry -3.59 rz 1.4 deg; joints [6.97, -132.208, -68.259, -60.695, 93.599, 1.618]
  MoveL 940 to (-45.45, -164.14, 367.42) mm, rotated rx -21.36 ry -3.51 rz 1.37 deg; joints [7.306, -131.477, -69.464, -60.248, 93.459, 1.95]
  MoveL 941 to (-45.18, -155.28, 363.77) mm, rotated rx -21.17 ry -2.81 rz 1.09 deg; joints [7.628, -130.107, -72.104, -58.81, 92.644, 2.267]
  MoveL 942 to (-45.02, -148.22, 360.78) mm, rotated rx -20.76 ry -2.28 rz 0.86 deg; joints [7.887, -128.905, -74.485, -57.241, 92.014, 2.519]
  MoveL 943 to (-44.95, -142.34, 357.87) mm, rotated rx -19.99 ry -1.94 rz 0.71 deg; joints [8.077, -127.683, -76.961, -55.233, 91.578, 2.7]
  MoveL 944 to (-45.38, -134.49, 355.56) mm, rotated rx -19.47 ry -1.46 rz 0.51 deg; joints [8.381, -126.513, -79.479, -53.4, 90.976, 2.993]
  MoveL 945 to (-44.5, -125.35, 353.1) mm, rotated rx -19.59 ry -1.26 rz 0.45 deg; joints [8.439, -125.584, -81.41, -52.529, 90.762, 3.051]
  MoveL 946 to (-45.24, -116.12, 351.18) mm, rotated rx -20.19 ry -1.54 rz 0.57 deg; joints [8.39, -124.958, -82.722, -52.424, 91.111, 3.009]
  MoveL 947 to (-43.96, -111.57, 349) mm, rotated rx -20.38 ry -1.73 rz 0.64 deg; joints [8.21, -124.489, -83.515, -52.276, 91.353, 2.834]
  MoveL 948 to (-44.99, -105.23, 346.11) mm, rotated rx -20.32 ry -2.11 rz 0.78 deg; joints [8.145, -123.696, -85.01, -51.492, 91.768, 2.769]
  MoveL 949 to (-44.76, -95.11, 340.98) mm, rotated rx -20.08 ry -2.39 rz 0.87 deg; joints [8.042, -122.322, -87.534, -50.088, 92.07, 2.667]
  MoveL 950 to (-47.43, -90.65, 339) mm, rotated rx -19.93 ry -2.21 rz 0.8 deg; joints [8.392, -121.674, -88.754, -49.369, 91.801, 3.009]
  MoveL 951 to (-40.46, -89.14, 340) mm, rotated rx -20.01 ry -2.4 rz 0.87 deg; joints [7.687, -121.833, -88.736, -49.313, 92.137, 2.316]
  MoveL 952 to (-45.1, -85.23, 338.05) mm, rotated rx -19.65 ry -2.24 rz 0.8 deg; joints [8.205, -121.123, -90.11, -48.288, 91.846, 2.823]
  MoveL 953 to (-45.03, -75.45, 334.4) mm, rotated rx -19.84 ry -2.23 rz 0.81 deg; joints [8.242, -120.127, -91.966, -47.611, 91.848, 2.861]
  MoveL 954 to (-45.2, -66.74, 331.1) mm, rotated rx -20.56 ry -2.23 rz 0.84 deg; joints [8.276, -119.46, -93.002, -47.968, 91.89, 2.901]
  MoveL 955 to (-44.35, -61.24, 329) mm, rotated rx -20.28 ry -2.25 rz 0.83 deg; joints [8.223, -118.769, -94.411, -46.97, 91.903, 2.847]
  MoveL 956 to (-45.09, -54.81, 326.55) mm, rotated rx -19.7 ry -2.08 rz 0.74 deg; joints [8.435, -117.836, -96.361, -45.377, 91.642, 3.049]
  MoveL 957 to (-44.93, -45.01, 322.7) mm, rotated rx -18.86 ry -1.85 rz 0.63 deg; joints [8.623, -116.474, -99.197, -43.08, 91.307, 3.225]
  MoveL 958 to (-44.89, -35.86, 320.51) mm, rotated rx -18.38 ry -1.91 rz 0.63 deg; joints [8.653, -115.534, -101.41, -41.32, 91.332, 3.249]
  MoveL 959 to (-46.04, -30.96, 318.79) mm, rotated rx -18.39 ry -1.88 rz 0.62 deg; joints [8.814, -115.031, -102.377, -40.861, 91.265, 3.406]
  MoveL 960 to (-45.22, -24.42, 316.35) mm, rotated rx -18.54 ry -1.96 rz 0.66 deg; joints [8.72, -114.436, -103.457, -40.522, 91.386, 3.317]
  MoveL 961 to (-44.97, -14.43, 313.72) mm, rotated rx -19.07 ry -2.04 rz 0.71 deg; joints [8.692, -113.749, -104.781, -40.41, 91.509, 3.295]
  MoveL 962 to (-44.81, -6.71, 310.57) mm, rotated rx -19.57 ry -1.89 rz 0.67 deg; joints [8.791, -113.082, -105.776, -40.591, 91.367, 3.398]
  MoveL 963 to (-45.17, -1.87, 308.47) mm, rotated rx -19.25 ry -1.72 rz 0.6 deg; joints [8.972, -112.437, -107.031, -39.673, 91.128, 3.571]
  MoveL 964 to (-45.05, 5.44, 306.23) mm, rotated rx -18.96 ry -1.55 rz 0.53 deg; joints [9.12, -111.67, -108.663, -38.529, 90.897, 3.714]
  MoveL 965 to (-44.91, 14.71, 303.12) mm, rotated rx -18.46 ry -1.22 rz 0.41 deg; joints [9.389, -110.627, -110.862, -36.897, 90.463, 3.97]
  MoveL 966 to (-45.38, 23.89, 300.54) mm, rotated rx -18.25 ry -0.9 rz 0.3 deg; joints [9.717, -109.749, -112.739, -35.712, 90.04, 4.288]
  MoveL 967 to (-44.13, 29.08, 299) mm, rotated rx -18.18 ry -1 rz 0.33 deg; joints [9.564, -109.309, -113.69, -35.121, 90.174, 4.137]
  MoveL 968 to (-45.15, 35.39, 296.22) mm, rotated rx -18.17 ry -0.84 rz 0.28 deg; joints [9.833, -108.604, -114.884, -34.637, 89.952, 4.4]
  MoveL 969 to (-44.94, 45.42, 291.99) mm, rotated rx -18.58 ry -0.83 rz 0.28 deg; joints [9.89, -107.669, -116.305, -34.562, 89.967, 4.462]
  MoveL 970 to (-43.29, 52.9, 290.66) mm, rotated rx -18.65 ry -0.88 rz 0.3 deg; joints [9.734, -107.208, -117.466, -33.932, 90.049, 4.311]
  MoveL 971 to (-45.82, 57.25, 288.63) mm, rotated rx -18.26 ry -0.87 rz 0.29 deg; joints [10.093, -106.59, -118.662, -32.957, 89.941, 4.657]
  MoveL 972 to (-44.97, 65.57, 286.35) mm, rotated rx -17.6 ry -0.89 rz 0.28 deg; joints [10.098, -105.783, -120.651, -31.121, 89.905, 4.649]
  MoveL 973 to (-45.11, 75.39, 283.42) mm, rotated rx -17.81 ry -0.74 rz 0.24 deg; joints [10.306, -104.987, -122.155, -30.64, 89.719, 4.857]
  MoveL 974 to (-45.09, 83.41, 280.89) mm, rotated rx -17.39 ry -0.88 rz 0.28 deg; joints [10.325, -104.227, -123.876, -29.241, 89.82, 4.867]
  MoveL 975 to (-45.74, 88.56, 278.75) mm, rotated rx -17.14 ry -0.96 rz 0.3 deg; joints [10.422, -103.657, -124.981, -28.457, 89.865, 4.957]
  MoveL 976 to (-45.92, 92.88, 278.43) mm, rotated rx -17.04 ry -0.93 rz 0.29 deg; joints [10.519, -103.433, -125.772, -27.79, 89.799, 5.05]
  MoveL 977 to (-32.23, -260.08, 404) mm, rotated rx -16.06 ry -1.34 rz 0.39 deg; joints [7.081, -142.871, -48.187, -64.954, 90.964, 1.693]
  MoveL 978 to (-33.79, -253.64, 402.33) mm, rotated rx -17.5 ry -1.53 rz 0.48 deg; joints [7.111, -142.869, -47.864, -66.707, 91.208, 1.732]
  MoveL 979 to (-35.53, -248.7, 400.85) mm, rotated rx -18.48 ry -1.68 rz 0.56 deg; joints [7.171, -142.757, -47.861, -67.795, 91.393, 1.797]
  MoveL 980 to (-35.19, -242.9, 398.42) mm, rotated rx -19.78 ry -1.72 rz 0.62 deg; joints [7.125, -142.708, -47.57, -69.435, 91.498, 1.76]
  MoveL 981 to (-35.22, -235.29, 396.02) mm, rotated rx -21.39 ry -1.93 rz 0.76 deg; joints [7.034, -142.693, -47.273, -71.347, 91.808, 1.679]
  MoveL 982 to (-34.82, -225.49, 391.72) mm, rotated rx -22.82 ry -2.17 rz 0.91 deg; joints [6.906, -142.036, -48.189, -72.507, 92.152, 1.558]
  MoveL 983 to (-35.15, -215.6, 386.7) mm, rotated rx -22.49 ry -2.4 rz 1 deg; joints [6.862, -139.904, -52.362, -70.129, 92.393, 1.514]
  MoveL 984 to (-35.03, -205.34, 382.65) mm, rotated rx -21.17 ry -2.09 rz 0.81 deg; joints [7.029, -137.252, -57.93, -65.905, 91.97, 1.673]
  MoveL 985 to (-34.82, -198.13, 380.35) mm, rotated rx -20.1 ry -2.07 rz 0.76 deg; joints [7.056, -135.527, -61.712, -62.775, 91.898, 1.694]
  MoveL 986 to (-34.65, -193.21, 378.5) mm, rotated rx -19.64 ry -2.09 rz 0.75 deg; joints [7.053, -134.547, -63.792, -61.218, 91.901, 1.69]
  MoveL 987 to (-34.92, -185.04, 375.22) mm, rotated rx -19.54 ry -2.24 rz 0.79 deg; joints [7.034, -133.33, -66.215, -59.907, 92.053, 1.67]
  MoveL 988 to (-35.24, -174.67, 371.98) mm, rotated rx -20.5 ry -2.91 rz 1.09 deg; joints [6.775, -132.578, -67.585, -60.224, 92.854, 1.421]
  MoveL 989 to (-35.57, -167.24, 370.46) mm, rotated rx -21.05 ry -3.21 rz 1.24 deg; joints [6.671, -132.053, -68.699, -60.182, 93.224, 1.32]
  MoveL 990 to (-34.02, -162.76, 368.18) mm, rotated rx -21.56 ry -3.15 rz 1.24 deg; joints [6.578, -131.684, -69.197, -60.567, 93.193, 1.23]
  MoveL 991 to (-35.03, -155.72, 364.6) mm, rotated rx -22.06 ry -3.14 rz 1.27 deg; joints [6.663, -130.906, -70.452, -60.585, 93.199, 1.316]
  MoveL 992 to (-34.19, -147.31, 360.9) mm, rotated rx -21.53 ry -2.55 rz 1 deg; joints [6.892, -129.419, -73.384, -58.621, 92.5, 1.54]
  MoveL 993 to (-36.19, -142.16, 358.29) mm, rotated rx -20.7 ry -2.01 rz 0.76 deg; joints [7.325, -128.192, -75.865, -56.553, 91.816, 1.963]
  MoveL 994 to (-34.9, -135.14, 355.82) mm, rotated rx -19.83 ry -1.68 rz 0.61 deg; joints [7.408, -126.92, -78.618, -54.218, 91.412, 2.04]
  MoveL 995 to (-34.82, -125.64, 352.33) mm, rotated rx -19.66 ry -1.61 rz 0.57 deg; joints [7.471, -125.706, -81.05, -52.827, 91.313, 2.1]
  MoveL 996 to (-36.56, -117.89, 350.48) mm, rotated rx -19.86 ry -1.54 rz 0.56 deg; joints [7.665, -124.975, -82.583, -52.225, 91.221, 2.293]
  MoveL 997 to (-34.13, -113.49, 348.27) mm, rotated rx -19.86 ry -1.79 rz 0.64 deg; joints [7.363, -124.459, -83.517, -51.803, 91.531, 1.995]
  MoveL 998 to (-34.89, -104.8, 344.69) mm, rotated rx -19.83 ry -2.13 rz 0.77 deg; joints [7.293, -123.433, -85.484, -50.814, 91.903, 1.927]
  MoveL 999 to (-35.29, -94.84, 341.43) mm, rotated rx -20.15 ry -2.41 rz 0.88 deg; joints [7.212, -122.522, -87.249, -50.276, 92.235, 1.849]
  MoveL 1000 to (-33.93, -88.08, 340) mm, rotated rx -20.08 ry -2.56 rz 0.93 deg; joints [7.041, -121.905, -88.678, -49.392, 92.417, 1.68]
  MoveL 1001 to (-35.62, -83.72, 338.17) mm, rotated rx -19.63 ry -2.48 rz 0.88 deg; joints [7.253, -121.187, -90.164, -48.167, 92.272, 1.886]
  MoveL 1002 to (-34.91, -75.43, 335.06) mm, rotated rx -19.53 ry -2.6 rz 0.92 deg; joints [7.154, -120.272, -91.976, -47.17, 92.42, 1.788]
  MoveL 1003 to (-34.69, -65.72, 330.89) mm, rotated rx -20.71 ry -2.75 rz 1.04 deg; joints [7.063, -119.634, -92.731, -48.229, 92.646, 1.705]
  MoveL 1004 to (-37.26, -61.15, 329) mm, rotated rx -20.54 ry -2.57 rz 0.96 deg; joints [7.407, -118.993, -93.956, -47.464, 92.389, 2.044]
  MoveL 1005 to (-31.94, -58.92, 330) mm, rotated rx -20.67 ry -2.52 rz 0.95 deg; joints [6.944, -119.107, -94.049, -47.416, 92.427, 1.588]
  MoveL 1006 to (-35.39, -54.86, 327.8) mm, rotated rx -20.08 ry -2.31 rz 0.85 deg; joints [7.399, -118.294, -95.644, -46.033, 92.097, 2.032]
  MoveL 1007 to (-34.98, -45.1, 323.58) mm, rotated rx -19.1 ry -2 rz 0.69 deg; joints [7.589, -116.826, -98.653, -43.525, 91.675, 2.213]
  MoveL 1008 to (-35.15, -34.9, 320.88) mm, rotated rx -18.46 ry -1.8 rz 0.6 deg; joints [7.77, -115.683, -101.267, -41.424, 91.395, 2.385]
  MoveL 1009 to (-36.71, -30.28, 319) mm, rotated rx -18.46 ry -1.79 rz 0.6 deg; joints [7.944, -115.171, -102.204, -40.998, 91.358, 2.555]
  MoveL 1010 to (-34.9, -24.27, 317.08) mm, rotated rx -18.35 ry -1.76 rz 0.58 deg; joints [7.813, -114.594, -103.413, -40.258, 91.346, 2.426]
  MoveL 1011 to (-35.18, -14.36, 313.56) mm, rotated rx -19.11 ry -1.86 rz 0.65 deg; joints [7.808, -113.862, -104.549, -40.603, 91.493, 2.428]
  MoveL 1012 to (-34.62, -6.23, 310.79) mm, rotated rx -19.53 ry -1.99 rz 0.71 deg; joints [7.705, -113.239, -105.632, -40.562, 91.668, 2.33]
  MoveL 1013 to (-35.68, -1.52, 309) mm, rotated rx -19.58 ry -1.98 rz 0.7 deg; joints [7.84, -112.76, -106.501, -40.215, 91.633, 2.463]
  MoveL 1014 to (-35.02, 5.26, 306.74) mm, rotated rx -19.25 ry -1.7 rz 0.59 deg; joints [7.974, -112.001, -108.083, -39.077, 91.299, 2.591]
  MoveL 1015 to (-34.93, 14.84, 302.35) mm, rotated rx -18.73 ry -1.64 rz 0.56 deg; joints [8.066, -110.79, -110.374, -37.48, 91.19, 2.677]
  MoveL 1016 to (-35.56, 22.54, 300.28) mm, rotated rx -18.42 ry -1.63 rz 0.54 deg; joints [8.194, -110.049, -112.055, -36.225, 91.129, 2.8]
  MoveL 1017 to (-34, 27.54, 298.56) mm, rotated rx -18.41 ry -1.56 rz 0.52 deg; joints [8.094, -109.599, -112.929, -35.797, 91.077, 2.701]
  MoveL 1018 to (-35.11, 35.36, 296.53) mm, rotated rx -18.26 ry -1.46 rz 0.48 deg; joints [8.328, -108.898, -114.478, -34.801, 90.912, 2.929]
  MoveL 1019 to (-34.87, 44.95, 293.08) mm, rotated rx -18.63 ry -1.25 rz 0.42 deg; joints [8.479, -108.065, -115.861, -34.63, 90.684, 3.081]
  MoveL 1020 to (-35.26, 53.51, 291.24) mm, rotated rx -18.55 ry -1.3 rz 0.44 deg; joints [8.544, -107.423, -117.393, -33.664, 90.726, 3.143]
  MoveL 1021 to (-34.6, 58.92, 288.59) mm, rotated rx -18.23 ry -1.28 rz 0.42 deg; joints [8.533, -106.744, -118.642, -32.773, 90.683, 3.129]
  MoveL 1022 to (-34.91, 65.73, 286.63) mm, rotated rx -17.77 ry -1.17 rz 0.38 deg; joints [8.704, -106.06, -120.233, -31.417, 90.508, 3.29]
  MoveL 1023 to (-34.98, 75.1, 282.97) mm, rotated rx -17.71 ry -1.05 rz 0.33 deg; joints [8.872, -105.115, -121.934, -30.603, 90.335, 3.454]
  MoveL 1024 to (-35.87, 82.6, 280.61) mm, rotated rx -17.36 ry -0.86 rz 0.27 deg; joints [9.187, -104.362, -123.563, -29.391, 90.045, 3.757]
  MoveL 1025 to (-38.82, 88.11, 279) mm, rotated rx -17.29 ry -0.81 rz 0.25 deg; joints [9.641, -103.84, -124.628, -28.782, 89.893, 4.198]
  MoveL 1026 to (-39.21, 90.55, 279) mm, rotated rx -17.26 ry -0.86 rz 0.27 deg; joints [9.678, -103.752, -125.041, -28.426, 89.934, 4.233]
  MoveL 1027 to (-26.43, -260.08, 404) mm, rotated rx -15.65 ry -1.24 rz 0.35 deg; joints [6.717, -142.662, -48.753, -64.193, 90.934, 1.337]
  MoveL 1028 to (-24.93, -254.7, 402.29) mm, rotated rx -16.46 ry -1.4 rz 0.41 deg; joints [6.547, -142.376, -49.129, -64.909, 91.172, 1.176]
  MoveL 1029 to (-25.66, -248.85, 400.31) mm, rotated rx -17.75 ry -1.59 rz 0.51 deg; joints [6.519, -142.332, -48.86, -66.514, 91.414, 1.156]
  MoveL 1030 to (-24.79, -243.96, 398.74) mm, rotated rx -19.07 ry -1.67 rz 0.58 deg; joints [6.419, -142.518, -48.157, -68.343, 91.556, 1.063]
  MoveL 1031 to (-24.94, -235.95, 397.15) mm, rotated rx -20.71 ry -1.87 rz 0.71 deg; joints [6.344, -142.556, -47.862, -70.24, 91.828, 0.995]
  MoveL 1032 to (-24.81, -226.11, 392.55) mm, rotated rx -22.23 ry -2.47 rz 1.01 deg; joints [6.087, -141.962, -48.597, -71.599, 92.561, 0.745]
  MoveL 1033 to (-25.19, -215.6, 386.85) mm, rotated rx -22.3 ry -2.96 rz 1.21 deg; joints [5.928, -140.028, -52.239, -69.957, 93.105, 0.587]
  MoveL 1034 to (-25.01, -205.23, 382.45) mm, rotated rx -21.49 ry -3 rz 1.18 deg; joints [5.917, -137.708, -57.001, -66.705, 93.125, 0.575]
  MoveL 1035 to (-24.19, -197.06, 380.81) mm, rotated rx -20.31 ry -2.93 rz 1.08 deg; joints [5.904, -135.871, -61.183, -63.183, 93.019, 0.56]
  MoveL 1036 to (-25.76, -192.31, 378.67) mm, rotated rx -19.73 ry -2.61 rz 0.94 deg; joints [6.167, -134.735, -63.525, -61.406, 92.615, 0.818]
  MoveL 1037 to (-25.12, -184.67, 375.92) mm, rotated rx -19.39 ry -2.43 rz 0.85 deg; joints [6.209, -133.473, -66.14, -59.716, 92.403, 0.858]
  MoveL 1038 to (-24.86, -174.65, 372.66) mm, rotated rx -20.07 ry -2.44 rz 0.89 deg; joints [6.187, -132.54, -67.881, -59.582, 92.442, 0.839]
  MoveL 1039 to (-23.76, -168.26, 370.6) mm, rotated rx -20.81 ry -2.42 rz 0.92 deg; joints [6.109, -132.142, -68.518, -60.09, 92.456, 0.763]
  MoveL 1040 to (-25.41, -163.58, 367.96) mm, rotated rx -21.38 ry -2.49 rz 0.98 deg; joints [6.203, -131.708, -69.087, -60.513, 92.539, 0.857]
  MoveL 1041 to (-24.98, -154.53, 364.33) mm, rotated rx -22.2 ry -2.49 rz 1.02 deg; joints [6.17, -130.944, -70.347, -60.843, 92.571, 0.827]
  MoveL 1042 to (-25.3, -145.3, 361) mm, rotated rx -22.02 ry -2.41 rz 0.97 deg; joints [6.248, -129.648, -72.958, -59.345, 92.458, 0.904]
  MoveL 1043 to (-24.09, -141.04, 359) mm, rotated rx -21.27 ry -2.31 rz 0.9 deg; joints [6.213, -128.687, -74.975, -57.546, 92.331, 0.868]
  MoveL 1044 to (-24.47, -134.81, 356.63) mm, rotated rx -20.03 ry -2.15 rz 0.78 deg; joints [6.34, -127.29, -78.05, -54.629, 92.105, 0.989]
  MoveL 1045 to (-25.46, -125.02, 352.53) mm, rotated rx -19.66 ry -2.02 rz 0.72 deg; joints [6.501, -125.872, -80.854, -52.874, 91.931, 1.147]
  MoveL 1046 to (-23.45, -116.48, 350.13) mm, rotated rx -19.99 ry -1.88 rz 0.69 deg; joints [6.409, -125.126, -82.343, -52.468, 91.81, 1.056]
  MoveL 1047 to (-27.32, -113.94, 348.58) mm, rotated rx -19.9 ry -1.82 rz 0.66 deg; joints [6.771, -124.653, -83.175, -52.007, 91.673, 1.413]
  MoveL 1048 to (-24.95, -105, 345.55) mm, rotated rx -19.67 ry -1.79 rz 0.64 deg; joints [6.606, -123.602, -85.353, -50.656, 91.664, 1.25]
  MoveL 1049 to (-25.02, -94.91, 341.55) mm, rotated rx -19.37 ry -2.52 rz 0.89 deg; joints [6.28, -122.398, -87.8, -49.099, 92.49, 0.928]
  MoveL 1050 to (-24.91, -87.38, 340.06) mm, rotated rx -19.62 ry -3.08 rz 1.1 deg; joints [6.004, -121.889, -88.986, -48.672, 93.137, 0.658]
  MoveL 1051 to (-25.28, -82.68, 339) mm, rotated rx -19.64 ry -3.15 rz 1.12 deg; joints [6.007, -121.468, -89.929, -48.169, 93.209, 0.661]
  MoveL 1052 to (-25.05, -74.92, 335.94) mm, rotated rx -19.78 ry -2.78 rz 1 deg; joints [6.178, -120.619, -91.467, -47.617, 92.794, 0.829]
  MoveL 1053 to (-25.4, -64.9, 331.35) mm, rotated rx -20.74 ry -2.49 rz 0.94 deg; joints [6.355, -119.771, -92.607, -48.291, 92.491, 1.006]
  MoveL 1054 to (-23.24, -60.46, 329) mm, rotated rx -20.92 ry -2.41 rz 0.92 deg; joints [6.207, -119.31, -93.311, -48.238, 92.43, 0.861]
  MoveL 1055 to (-29.78, -58.92, 330) mm, rotated rx -20.73 ry -2.51 rz 0.95 deg; joints [6.755, -119.163, -93.927, -47.551, 92.443, 1.401]
  MoveL 1056 to (-24.8, -55.06, 327.86) mm, rotated rx -20.57 ry -2.3 rz 0.86 deg; joints [6.418, -118.664, -94.809, -47.023, 92.27, 1.068]
  MoveL 1057 to (-25.04, -45.23, 324.49) mm, rotated rx -19.33 ry -2.07 rz 0.72 deg; joints [6.605, -117.193, -98.078, -43.993, 91.944, 1.247]
  MoveL 1058 to (-25.41, -37.01, 321) mm, rotated rx -18.76 ry -1.8 rz 0.61 deg; joints [6.813, -116.066, -100.337, -42.291, 91.603, 1.448]
  MoveL 1059 to (-24.77, -31.82, 318.71) mm, rotated rx -18.68 ry -1.51 rz 0.51 deg; joints [6.924, -115.445, -101.456, -41.725, 91.272, 1.557]
  MoveL 1060 to (-24.94, -24.35, 317.78) mm, rotated rx -18.49 ry -1.36 rz 0.45 deg; joints [7.048, -114.846, -103.032, -40.555, 91.08, 1.677]
  MoveL 1061 to (-24.92, -14.13, 313.97) mm, rotated rx -18.79 ry -1.43 rz 0.49 deg; joints [7.032, -113.925, -104.668, -40.142, 91.17, 1.663]
  MoveL 1062 to (-24.74, -5.36, 310.95) mm, rotated rx -19.53 ry -1.62 rz 0.58 deg; joints [6.915, -113.338, -105.558, -40.577, 91.424, 1.553]
  MoveL 1063 to (-26.22, -0.69, 309) mm, rotated rx -19.73 ry -1.64 rz 0.59 deg; joints [7.064, -112.883, -106.294, -40.484, 91.428, 1.7]
  MoveL 1064 to (-25.01, 5.43, 306.65) mm, rotated rx -19.33 ry -1.57 rz 0.55 deg; joints [7.012, -112.157, -107.794, -39.315, 91.34, 1.647]
  MoveL 1065 to (-25.02, 14.82, 303.67) mm, rotated rx -18.63 ry -1.63 rz 0.55 deg; joints [7.023, -111.111, -110.151, -37.304, 91.374, 1.654]
  MoveL 1066 to (-23.96, 23.35, 300.67) mm, rotated rx -18.64 ry -1.53 rz 0.52 deg; joints [6.997, -110.319, -111.663, -36.605, 91.275, 1.628]
  MoveL 1067 to (-26.4, 27.76, 298.83) mm, rotated rx -18.32 ry -1.52 rz 0.5 deg; joints [7.288, -109.732, -112.838, -35.685, 91.199, 1.911]
  MoveL 1068 to (-25.17, 35.58, 297.35) mm, rotated rx -18.19 ry -1.75 rz 0.58 deg; joints [7.041, -109.202, -114.234, -34.684, 91.486, 1.669]
  MoveL 1069 to (-24.97, 45.04, 293.71) mm, rotated rx -18.69 ry -1.86 rz 0.63 deg; joints [6.974, -108.427, -115.434, -34.761, 91.63, 1.606]
  MoveL 1070 to (-24.82, 53.04, 290.99) mm, rotated rx -18.53 ry -1.85 rz 0.62 deg; joints [6.995, -107.664, -116.975, -33.823, 91.607, 1.626]
  MoveL 1071 to (-25.46, 58.28, 288.82) mm, rotated rx -18.41 ry -1.79 rz 0.6 deg; joints [7.125, -107.086, -118.038, -33.216, 91.522, 1.752]
  MoveL 1072 to (-24.89, 65.15, 286.45) mm, rotated rx -17.89 ry -1.65 rz 0.53 deg; joints [7.19, -106.335, -119.696, -31.79, 91.338, 1.812]
  MoveL 1073 to (-25.49, 75.04, 283.81) mm, rotated rx -17.87 ry -1.43 rz 0.46 deg; joints [7.449, -105.518, -121.429, -30.866, 91.053, 2.066]
  MoveL 1074 to (-28.19, 81.77, 281.57) mm, rotated rx -17.13 ry -1.37 rz 0.42 deg; joints [7.88, -104.716, -123.315, -29.034, 90.859, 2.479]
  MoveL 1075 to (-17.45, -260.08, 404) mm, rotated rx -16.27 ry -1.01 rz 0.29 deg; joints [6.169, -143.282, -47.313, -65.65, 90.846, 0.808]
  MoveL 1076 to (-14.41, -255.53, 402.43) mm, rotated rx -16.67 ry -1.26 rz 0.38 deg; joints [5.862, -142.866, -48.067, -65.714, 91.18, 0.511]
  MoveL 1077 to (-14.58, -248.6, 400.47) mm, rotated rx -17.74 ry -1.51 rz 0.48 deg; joints [5.772, -142.523, -48.543, -66.642, 91.485, 0.425]
  MoveL 1078 to (-15.58, -243.43, 398.48) mm, rotated rx -19.03 ry -1.59 rz 0.55 deg; joints [5.806, -142.572, -48.067, -68.363, 91.583, 0.461]
  MoveL 1079 to (-15.09, -235.45, 396.54) mm, rotated rx -20.29 ry -1.76 rz 0.65 deg; joints [5.701, -142.274, -48.497, -69.488, 91.802, 0.359]
  MoveL 1080 to (-14.73, -225.26, 392.82) mm, rotated rx -21.72 ry -2.53 rz 1.01 deg; joints [5.359, -141.701, -49.355, -70.629, 92.71, 0.023]
  MoveL 1081 to (-15.21, -214.89, 387.25) mm, rotated rx -22.14 ry -2.85 rz 1.16 deg; joints [5.26, -140.065, -52.316, -69.721, 93.077, -0.075]
  MoveL 1082 to (-15.34, -205.47, 383.35) mm, rotated rx -21.47 ry -3.15 rz 1.24 deg; joints [5.149, -138.047, -56.483, -66.909, 93.405, -0.186]
  MoveL 1083 to (-15.71, -197.43, 380.62) mm, rotated rx -20.48 ry -3.2 rz 1.2 deg; joints [5.161, -136.2, -60.47, -63.779, 93.438, -0.173]
  MoveL 1084 to (-14.14, -192.85, 378.75) mm, rotated rx -20.13 ry -3.06 rz 1.12 deg; joints [5.104, -135.313, -62.307, -62.486, 93.292, -0.23]
  MoveL 1085 to (-14.53, -184.94, 376.09) mm, rotated rx -19.99 ry -2.64 rz 0.96 deg; joints [5.31, -134.08, -64.817, -61.066, 92.809, -0.027]
  MoveL 1086 to (-14.64, -174.7, 372.78) mm, rotated rx -20.31 ry -1.97 rz 0.73 deg; joints [5.604, -132.822, -67.269, -60.183, 92.052, 0.264]
  MoveL 1087 to (-14.54, -167.43, 371) mm, rotated rx -21.03 ry -1.69 rz 0.65 deg; joints [5.717, -132.314, -68.216, -60.466, 91.742, 0.377]
  MoveL 1088 to (-16.23, -162.65, 368.27) mm, rotated rx -21.49 ry -1.75 rz 0.69 deg; joints [5.819, -131.8, -68.961, -60.692, 91.803, 0.478]
  MoveL 1089 to (-14.9, -154.96, 365.09) mm, rotated rx -21.87 ry -1.76 rz 0.71 deg; joints [5.714, -130.984, -70.431, -60.421, 91.836, 0.374]
  MoveL 1090 to (-15.12, -145.6, 361) mm, rotated rx -21.88 ry -2.44 rz 0.98 deg; joints [5.433, -129.786, -72.736, -59.324, 92.604, 0.096]
  MoveL 1091 to (-15.04, -141.04, 359) mm, rotated rx -21.32 ry -2.66 rz 1.04 deg; joints [5.329, -128.913, -74.571, -57.799, 92.851, -0.007]
  MoveL 1092 to (-14.97, -134.78, 357.32) mm, rotated rx -20.3 ry -2.65 rz 0.98 deg; joints [5.338, -127.717, -77.316, -55.234, 92.815, 0.002]
  MoveL 1093 to (-15.27, -125.01, 353.45) mm, rotated rx -19.81 ry -2.31 rz 0.83 deg; joints [5.523, -126.25, -80.28, -53.243, 92.415, 0.184]
  MoveL 1094 to (-15.28, -115.43, 350.5) mm, rotated rx -20.06 ry -2.26 rz 0.82 deg; joints [5.55, -125.304, -82.161, -52.557, 92.357, 0.211]
  MoveL 1095 to (-14.84, -105.39, 347.33) mm, rotated rx -19.38 ry -2.32 rz 0.82 deg; joints [5.492, -123.949, -85.128, -50.271, 92.421, 0.153]
  MoveL 1096 to (-14.81, -95.31, 342.98) mm, rotated rx -18.77 ry -2.67 rz 0.91 deg; joints [5.327, -122.557, -87.969, -48.215, 92.812, -0.009]
  MoveL 1097 to (-14.7, -87.45, 340.33) mm, rotated rx -19.44 ry -2.61 rz 0.92 deg; joints [5.341, -121.98, -88.913, -48.513, 92.757, 0.005]
  MoveL 1098 to (-15.08, -82.61, 338.71) mm, rotated rx -19.85 ry -2.56 rz 0.92 deg; joints [5.394, -121.62, -89.508, -48.686, 92.706, 0.057]
  MoveL 1099 to (-14.96, -74.96, 336.13) mm, rotated rx -20.28 ry -2.28 rz 0.84 deg; joints [5.522, -120.958, -90.678, -48.61, 92.392, 0.183]
  MoveL 1100 to (-14.94, -64.59, 332.02) mm, rotated rx -20.81 ry -2.15 rz 0.82 deg; joints [5.586, -120.004, -92.297, -48.478, 92.25, 0.246]
  MoveL 1101 to (-15.02, -55.11, 327.84) mm, rotated rx -20.89 ry -2.14 rz 0.82 deg; joints [5.6, -118.944, -94.188, -47.727, 92.241, 0.261]
  MoveL 1102 to (-15.17, -45.18, 324.86) mm, rotated rx -19.68 ry -1.73 rz 0.62 deg; joints [5.85, -117.494, -97.474, -44.681, 91.733, 0.505]
  MoveL 1103 to (-14.85, -35.89, 321.13) mm, rotated rx -19.2 ry -1.28 rz 0.44 deg; joints [6.074, -116.291, -99.866, -43.007, 91.205, 0.725]
  MoveL 1104 to (-15.86, -30.83, 319) mm, rotated rx -18.93 ry -1.23 rz 0.42 deg; joints [6.206, -115.634, -101.16, -42.103, 91.127, 0.854]
  MoveL 1105 to (-14.96, -24.33, 317.49) mm, rotated rx -18.45 ry -1.19 rz 0.4 deg; joints [6.157, -114.955, -102.821, -40.647, 91.079, 0.804]
  MoveL 1106 to (-14.78, -14.2, 313.61) mm, rotated rx -18.61 ry -1.26 rz 0.43 deg; joints [6.11, -113.991, -104.575, -40.014, 91.17, 0.759]
  MoveL 1107 to (-15, -4.3, 311.09) mm, rotated rx -19.5 ry -1.28 rz 0.45 deg; joints [6.124, -113.429, -105.54, -40.494, 91.21, 0.774]
  MoveL 1108 to (-12.31, 1.36, 310) mm, rotated rx -19.44 ry -1.37 rz 0.48 deg; joints [5.808, -113.049, -106.512, -39.851, 91.357, 0.464]
  MoveL 1109 to (-15.18, 5.64, 307.3) mm, rotated rx -19.32 ry -1.65 rz 0.58 deg; joints [5.95, -112.424, -107.51, -39.349, 91.62, 0.603]
  MoveL 1110 to (-15.11, 14.82, 303.74) mm, rotated rx -18.7 ry -1.51 rz 0.51 deg; joints [6.044, -111.312, -109.81, -37.539, 91.442, 0.693]
  MoveL 1111 to (-14.88, 24.29, 301.08) mm, rotated rx -18.46 ry -1.59 rz 0.53 deg; joints [5.983, -110.469, -111.688, -36.27, 91.538, 0.634]
  MoveL 1112 to (-15.97, 29.45, 299) mm, rotated rx -18.13 ry -1.63 rz 0.53 deg; joints [6.089, -109.848, -112.959, -35.28, 91.553, 0.736]
  MoveL 1113 to (-15.18, 35.51, 297.46) mm, rotated rx -18.14 ry -1.55 rz 0.51 deg; joints [6.059, -109.381, -113.986, -34.741, 91.475, 0.707]
  MoveL 1114 to (-14.97, 44.98, 293.33) mm, rotated rx -18.6 ry -1.55 rz 0.52 deg; joints [6.046, -108.512, -115.263, -34.789, 91.484, 0.696]
  MoveL 1115 to (-14.69, 54.04, 291.13) mm, rotated rx -18.48 ry -1.5 rz 0.5 deg; joints [6.06, -107.793, -116.919, -33.734, 91.426, 0.709]
  MoveL 1116 to (-16.26, 58.68, 289) mm, rotated rx -18.6 ry -1.62 rz 0.54 deg; joints [6.17, -107.308, -117.664, -33.591, 91.534, 0.817]
  MoveL 1117 to (-14.96, 64.99, 286.7) mm, rotated rx -18.5 ry -1.54 rz 0.52 deg; joints [6.08, -106.714, -118.818, -32.936, 91.469, 0.729]
  MoveL 1118 to (-14.97, 73.52, 284.55) mm, rotated rx -18.23 ry -1.64 rz 0.54 deg; joints [6.033, -106.02, -120.477, -31.698, 91.576, 0.682]
  MoveL 1119 to (-4.57, -255.53, 402.27) mm, rotated rx -17 ry -1.92 rz 0.59 deg; joints [4.913, -143.425, -46.869, -66.705, 92.092, -0.413]
  MoveL 1120 to (-4.61, -247.85, 400.58) mm, rotated rx -18.28 ry -1.4 rz 0.46 deg; joints [5.113, -143.072, -47.356, -67.842, 91.509, -0.219]
  MoveL 1121 to (-6.02, -242.78, 398.56) mm, rotated rx -19.06 ry -1.23 rz 0.42 deg; joints [5.277, -142.686, -47.889, -68.473, 91.301, -0.059]
  MoveL 1122 to (-5.32, -235.34, 396.26) mm, rotated rx -19.79 ry -1.35 rz 0.49 deg; joints [5.175, -142.003, -49.148, -68.624, 91.458, -0.159]
  MoveL 1123 to (-5.16, -225.09, 392.67) mm, rotated rx -21.12 ry -1.87 rz 0.72 deg; joints [4.95, -141.331, -50.223, -69.56, 92.055, -0.382]
  MoveL 1124 to (-3.89, -217.84, 390.21) mm, rotated rx -21.69 ry -2.18 rz 0.87 deg; joints [4.727, -140.617, -51.579, -69.492, 92.429, -0.603]
  MoveL 1125 to (-5.76, -213.19, 388.27) mm, rotated rx -21.65 ry -2.51 rz 1 deg; joints [4.724, -139.786, -53.239, -68.627, 92.781, -0.606]
  MoveL 1126 to (-4.95, -205.12, 385.85) mm, rotated rx -21.21 ry -2.94 rz 1.14 deg; joints [4.485, -138.318, -56.413, -66.488, 93.272, -0.843]
  MoveL 1127 to (-4.51, -196.39, 381.46) mm, rotated rx -20.88 ry -2.76 rz 1.05 deg; joints [4.518, -136.617, -59.723, -64.543, 93.071, -0.809]
  MoveL 1128 to (-5.57, -191.98, 378.8) mm, rotated rx -20.61 ry -2.42 rz 0.91 deg; joints [4.735, -135.62, -61.604, -63.388, 92.67, -0.594]
  MoveL 1129 to (-5.17, -185.29, 376.98) mm, rotated rx -20.64 ry -1.78 rz 0.67 deg; joints [4.968, -134.677, -63.548, -62.406, 91.957, -0.364]
  MoveL 1130 to (-4.9, -174.91, 373.2) mm, rotated rx -20.84 ry -1.06 rz 0.4 deg; joints [5.254, -133.27, -66.279, -61.275, 91.136, -0.081]
  MoveL 1131 to (-4.87, -166.78, 370.33) mm, rotated rx -21.26 ry -0.86 rz 0.34 deg; joints [5.334, -132.398, -67.917, -60.928, 90.919, -0.003]
  MoveL 1132 to (-4.37, -162.33, 369) mm, rotated rx -21.46 ry -0.85 rz 0.33 deg; joints [5.303, -131.961, -68.783, -60.708, 90.905, -0.033]
  MoveL 1133 to (-4.91, -155.14, 365.86) mm, rotated rx -21.43 ry -1.04 rz 0.41 deg; joints [5.261, -130.957, -70.711, -59.751, 91.115, -0.075]
  MoveL 1134 to (-5.22, -144.7, 361.11) mm, rotated rx -21.01 ry -1.71 rz 0.65 deg; joints [4.983, -129.378, -73.835, -57.789, 91.874, -0.349]
  MoveL 1135 to (-5.26, -135.06, 357.87) mm, rotated rx -20.41 ry -2.16 rz 0.8 deg; joints [4.776, -127.983, -76.837, -55.588, 92.39, -0.553]
  MoveL 1136 to (-5.12, -125.35, 354.41) mm, rotated rx -20 ry -2 rz 0.73 deg; joints [4.832, -126.629, -79.637, -53.732, 92.206, -0.497]
  MoveL 1137 to (-5.09, -116.06, 351.13) mm, rotated rx -19.92 ry -2.03 rz 0.73 deg; joints [4.81, -125.53, -81.85, -52.538, 92.238, -0.518]
  MoveL 1138 to (-5.02, -105.52, 347.07) mm, rotated rx -19.42 ry -2.2 rz 0.77 deg; joints [4.715, -124.119, -84.758, -50.546, 92.434, -0.612]
  MoveL 1139 to (-4.96, -95.43, 343.44) mm, rotated rx -18.89 ry -1.88 rz 0.64 deg; joints [4.854, -122.755, -87.601, -48.525, 92.073, -0.474]
  MoveL 1140 to (-4.4, -86.34, 340.65) mm, rotated rx -19.65 ry -1.54 rz 0.55 deg; joints [4.965, -122.095, -88.725, -48.822, 91.692, -0.366]
  MoveL 1141 to (-5.6, -81.42, 338.93) mm, rotated rx -20.07 ry -1.62 rz 0.59 deg; joints [5.025, -121.725, -89.324, -49.016, 91.774, -0.307]
  MoveL 1142 to (-5.09, -74.67, 336.83) mm, rotated rx -20.49 ry -1.54 rz 0.57 deg; joints [5.017, -121.204, -90.278, -48.998, 91.686, -0.315]
  MoveL 1143 to (-4.99, -64.47, 332.37) mm, rotated rx -20.68 ry -1.51 rz 0.57 deg; joints [5.016, -120.1, -92.23, -48.34, 91.66, -0.317]
  MoveL 1144 to (-3.76, -58.63, 330) mm, rotated rx -20.7 ry -1.61 rz 0.61 deg; joints [4.849, -119.501, -93.353, -47.847, 91.795, -0.481]
  MoveL 1145 to (-5.52, -54.36, 328.06) mm, rotated rx -20.73 ry -1.85 rz 0.7 deg; joints [4.885, -119.011, -94.228, -47.487, 92.041, -0.446]
  MoveL 1146 to (-5.12, -45.28, 324.88) mm, rotated rx -20.27 ry -1.76 rz 0.65 deg; joints [4.888, -117.911, -96.522, -45.836, 91.943, -0.442]
  MoveL 1147 to (-4.86, -34.92, 321.07) mm, rotated rx -19.57 ry -1.27 rz 0.45 deg; joints [5.122, -116.547, -99.355, -43.657, 91.373, -0.211]
  MoveL 1148 to (-8.36, -30.28, 319) mm, rotated rx -19.03 ry -0.99 rz 0.34 deg; joints [5.609, -115.749, -100.974, -42.285, 90.989, 0.267]
  MoveL 1149 to (-5.01, -24.38, 318.11) mm, rotated rx -18.52 ry -0.82 rz 0.27 deg; joints [5.382, -115.206, -102.474, -40.826, 90.842, 0.045]
  MoveL 1150 to (-4.95, -14.22, 314.03) mm, rotated rx -18.54 ry -0.78 rz 0.26 deg; joints [5.398, -114.16, -104.395, -39.975, 90.798, 0.06]
  MoveL 1151 to (-4.9, -4.33, 311.18) mm, rotated rx -19.18 ry -0.97 rz 0.34 deg; joints [5.285, -113.506, -105.574, -40.083, 91.025, -0.051]
  MoveL 1152 to (-6.39, 1.94, 310) mm, rotated rx -19.17 ry -1.24 rz 0.43 deg; joints [5.281, -113.042, -106.706, -39.405, 91.312, -0.055]
  MoveL 1153 to (-4.58, 6.25, 307.41) mm, rotated rx -19.14 ry -1.21 rz 0.42 deg; joints [5.111, -112.517, -107.512, -39.102, 91.312, -0.222]
  MoveL 1154 to (-5.18, 14.82, 303.69) mm, rotated rx -18.81 ry -1.24 rz 0.42 deg; joints [5.151, -111.509, -109.43, -37.859, 91.34, -0.182]
  MoveL 1155 to (-5.14, 24.94, 301.22) mm, rotated rx -18.41 ry -1.09 rz 0.36 deg; joints [5.233, -110.585, -111.606, -36.209, 91.166, -0.102]
  MoveL 1156 to (-5.2, 35.14, 297.62) mm, rotated rx -18.16 ry -1.05 rz 0.35 deg; joints [5.263, -109.57, -113.659, -34.923, 91.115, -0.072]
  MoveL 1157 to (-4.9, 44.7, 294.41) mm, rotated rx -18.61 ry -1.15 rz 0.39 deg; joints [5.167, -108.846, -114.906, -34.847, 91.239, -0.167]
  MoveL 1158 to (-5.16, 54.21, 291.45) mm, rotated rx -18.38 ry -1.24 rz 0.41 deg; joints [5.135, -107.985, -116.75, -33.638, 91.341, -0.198]
  MoveL 1159 to (-2.66, 58.68, 289) mm, rotated rx -18.26 ry -1.32 rz 0.44 deg; joints [4.794, -107.493, -117.557, -33.213, 91.494, -0.532]
  MoveL 1160 to (-4.96, 64.5, 287.78) mm, rotated rx -18.28 ry -1.49 rz 0.49 deg; joints [4.943, -107.063, -118.571, -32.636, 91.645, -0.386]
  MoveL 1161 to (-4.84, 73.58, 285.66) mm, rotated rx -18.01 ry -1.61 rz 0.52 deg; joints [4.846, -106.371, -120.3, -31.334, 91.785, -0.48]
  MoveL 1162 to (1.03, -260.08, 404) mm, rotated rx -17.5 ry -3.16 rz 1 deg; joints [4.051, -145.048, -43.52, -68.969, 93.58, -1.258]
  MoveL 1163 to (4.67, -254.08, 403.13) mm, rotated rx -19.04 ry -3.19 rz 1.1 deg; joints [3.781, -145.474, -42.432, -71.192, 93.658, -1.53]
  MoveL 1164 to (5.36, -245.42, 400.97) mm, rotated rx -20.03 ry -2.36 rz 0.86 deg; joints [4.041, -144.627, -43.997, -71.435, 92.728, -1.277]
  MoveL 1165 to (4.66, -240.18, 399) mm, rotated rx -19.79 ry -1.87 rz 0.67 deg; joints [4.272, -143.327, -46.664, -69.817, 92.172, -1.048]
  MoveL 1166 to (5.17, -235.12, 397.5) mm, rotated rx -19.9 ry -1.57 rz 0.57 deg; joints [4.349, -142.499, -48.354, -69.054, 91.839, -0.973]
  MoveL 1167 to (5.1, -225.16, 392.8) mm, rotated rx -20.61 ry -1.4 rz 0.53 deg; joints [4.413, -141.152, -50.736, -68.731, 91.634, -0.911]
  MoveL 1168 to (4.67, -217.5, 390.21) mm, rotated rx -20.97 ry -2.03 rz 0.78 deg; joints [4.18, -140.227, -52.576, -68.184, 92.345, -1.143]
  MoveL 1169 to (5.41, -212.92, 388.76) mm, rotated rx -21.05 ry -2.39 rz 0.92 deg; joints [3.971, -139.636, -53.804, -67.647, 92.769, -1.35]
  MoveL 1170 to (5.01, -205.09, 385.95) mm, rotated rx -20.83 ry -2.72 rz 1.03 deg; joints [3.853, -138.281, -56.618, -65.975, 93.133, -1.466]
  MoveL 1171 to (5.07, -194.85, 381.54) mm, rotated rx -21.79 ry -2.41 rz 0.96 deg; joints [3.958, -137.232, -58.372, -66.223, 92.78, -1.365]
  MoveL 1172 to (0.47, -190.5, 379) mm, rotated rx -21.32 ry -1.85 rz 0.72 deg; joints [4.523, -135.986, -60.796, -64.545, 92.099, -0.804]
  MoveL 1173 to (4.92, -185.21, 378.3) mm, rotated rx -21.73 ry -1.1 rz 0.44 deg; joints [4.506, -135.616, -61.608, -64.514, 91.293, -0.822]
  MoveL 1174 to (4.86, -175.37, 374.17) mm, rotated rx -21.16 ry -0.33 rz 0.13 deg; joints [4.826, -133.726, -65.425, -62.004, 90.426, -0.504]
  MoveL 1175 to (4.54, -166.93, 370.36) mm, rotated rx -21.17 ry -0.42 rz 0.16 deg; joints [4.807, -132.507, -67.739, -60.918, 90.523, -0.524]
  MoveL 1176 to (5.44, -162.65, 369) mm, rotated rx -21.29 ry -0.56 rz 0.22 deg; joints [4.673, -132.062, -68.638, -60.586, 90.692, -0.655]
  MoveL 1177 to (4.96, -155.17, 366.02) mm, rotated rx -21.03 ry -0.82 rz 0.32 deg; joints [4.586, -130.942, -70.9, -59.191, 90.992, -0.742]
  MoveL 1178 to (5.17, -144.9, 361.59) mm, rotated rx -20.56 ry -1.24 rz 0.46 deg; joints [4.371, -129.376, -74.049, -57.139, 91.47, -0.953]
  MoveL 1179 to (4.9, -134.7, 357.67) mm, rotated rx -20.35 ry -1.36 rz 0.5 deg; joints [4.321, -128.015, -76.778, -55.57, 91.611, -1.001]
  MoveL 1180 to (5.32, -124.68, 354.31) mm, rotated rx -20.24 ry -1.15 rz 0.42 deg; joints [4.37, -126.784, -79.287, -54.175, 91.378, -0.953]
  MoveL 1181 to (4.65, -115.43, 351.06) mm, rotated rx -19.74 ry -1.16 rz 0.42 deg; joints [4.402, -125.491, -82.007, -52.251, 91.394, -0.92]
  MoveL 1182 to (4.96, -105.53, 347.09) mm, rotated rx -19.43 ry -1.39 rz 0.49 deg; joints [4.25, -124.231, -84.538, -50.677, 91.669, -1.069]
  MoveL 1183 to (4.92, -95.52, 343.76) mm, rotated rx -19.37 ry -1.21 rz 0.42 deg; joints [4.326, -123.108, -86.813, -49.457, 91.459, -0.993]
  MoveL 1184 to (4.61, -86.18, 340.92) mm, rotated rx -19.69 ry -1.07 rz 0.38 deg; joints [4.409, -122.259, -88.469, -48.97, 91.293, -0.913]
  MoveL 1185 to (5.68, -80.57, 339) mm, rotated rx -19.98 ry -1.11 rz 0.4 deg; joints [4.287, -121.806, -89.296, -48.883, 91.355, -1.034]
  MoveL 1186 to (4.81, -74.22, 336.78) mm, rotated rx -20.45 ry -1.25 rz 0.47 deg; joints [4.286, -121.322, -90.114, -49.03, 91.498, -1.036]
  MoveL 1187 to (5.1, -64.47, 332.2) mm, rotated rx -20.61 ry -1.16 rz 0.44 deg; joints [4.289, -120.215, -92.033, -48.368, 91.399, -1.034]
  MoveL 1188 to (5.68, -57.67, 330.31) mm, rotated rx -20.54 ry -1.06 rz 0.4 deg; joints [4.278, -119.543, -93.466, -47.541, 91.292, -1.044]
  MoveL 1189 to (4.64, -53.22, 328.48) mm, rotated rx -20.58 ry -1.12 rz 0.42 deg; joints [4.33, -119.055, -94.36, -47.174, 91.356, -0.993]
  MoveL 1190 to (5.08, -45.36, 325.47) mm, rotated rx -20.24 ry -1.22 rz 0.45 deg; joints [4.224, -118.121, -96.26, -45.873, 91.478, -1.097]
  MoveL 1191 to (5.02, -34.71, 321.37) mm, rotated rx -20 ry -1.32 rz 0.48 deg; joints [4.153, -116.934, -98.6, -44.479, 91.602, -1.166]
  MoveL 1192 to (4.96, -24.34, 317.58) mm, rotated rx -19.03 ry -0.85 rz 0.29 deg; joints [4.387, -115.511, -101.656, -41.869, 91.074, -0.933]
  MoveL 1193 to (4.91, -14.24, 314.4) mm, rotated rx -18.5 ry -0.44 rz 0.15 deg; joints [4.601, -114.364, -104.148, -39.986, 90.602, -0.721]
  MoveL 1194 to (4.87, -4.34, 311.6) mm, rotated rx -18.99 ry -0.57 rz 0.19 deg; joints [4.524, -113.663, -105.478, -39.846, 90.745, -0.797]
  MoveL 1195 to (4.94, 5.45, 307.27) mm, rotated rx -19.11 ry -0.61 rz 0.21 deg; joints [4.477, -112.659, -107.194, -39.256, 90.798, -0.844]
  MoveL 1196 to (5.19, 14.87, 304.09) mm, rotated rx -18.92 ry -0.65 rz 0.22 deg; joints [4.411, -111.743, -109.074, -38.099, 90.856, -0.909]
  MoveL 1197 to (5.21, 24.31, 301.56) mm, rotated rx -18.58 ry -0.63 rz 0.21 deg; joints [4.399, -110.878, -111.056, -36.651, 90.845, -0.919]
  MoveL 1198 to (4.28, 29.45, 299) mm, rotated rx -18.16 ry -0.69 rz 0.23 deg; joints [4.453, -110.175, -112.411, -35.577, 90.9, -0.866]
  MoveL 1199 to (5.19, 35.28, 297.31) mm, rotated rx -18.12 ry -0.69 rz 0.23 deg; joints [4.341, -109.699, -113.44, -34.978, 90.925, -0.974]
  MoveL 1200 to (4.81, 44.9, 294.54) mm, rotated rx -18.35 ry -0.84 rz 0.28 deg; joints [4.275, -108.975, -114.885, -34.492, 91.09, -1.04]
  MoveL 1201 to (5.11, 54.34, 291.51) mm, rotated rx -18.24 ry -1.11 rz 0.37 deg; joints [4.046, -108.182, -116.552, -33.517, 91.425, -1.264]
  MoveL 1202 to (1.87, 58.68, 289) mm, rotated rx -18.2 ry -1.2 rz 0.4 deg; joints [4.348, -107.571, -117.474, -33.162, 91.46, -0.969]
  MoveL 1203 to (4.87, 64.48, 287.96) mm, rotated rx -18.15 ry -1.08 rz 0.36 deg; joints [4.064, -107.243, -118.389, -32.535, 91.392, -1.246]
  MoveL 1204 to (5.15, 74.75, 284.89) mm, rotated rx -18.18 ry -1 rz 0.33 deg; joints [4.058, -106.408, -120.105, -31.682, 91.306, -1.252]
  MoveL 1205 to (5.16, 81.13, 283) mm, rotated rx -17.8 ry -0.98 rz 0.32 deg; joints [4.049, -105.815, -121.508, -30.495, 91.294, -1.259]
  MoveL 1206 to (14.28, -251.67, 402.7) mm, rotated rx -19.97 ry -2.99 rz 1.09 deg; joints [3.193, -146.16, -40.882, -73.015, 93.549, -2.114]
  MoveL 1207 to (14.85, -245.16, 401) mm, rotated rx -20.68 ry -2.87 rz 1.08 deg; joints [3.189, -145.559, -42.023, -73.18, 93.409, -2.123]
  MoveL 1208 to (16.66, -240.18, 399) mm, rotated rx -20.78 ry -2.71 rz 1.03 deg; joints [3.114, -144.661, -43.795, -72.404, 93.247, -2.197]
  MoveL 1209 to (15.03, -234.31, 396.4) mm, rotated rx -20.82 ry -2.44 rz 0.93 deg; joints [3.316, -143.427, -46.202, -71.259, 92.928, -1.997]
  MoveL 1210 to (15.22, -224.6, 391.97) mm, rotated rx -20.25 ry -2.35 rz 0.87 deg; joints [3.31, -141.137, -50.846, -68.336, 92.84, -2]
  MoveL 1211 to (15.29, -217.82, 390.7) mm, rotated rx -20.43 ry -2.44 rz 0.91 deg; joints [3.254, -140.28, -52.72, -67.497, 92.939, -2.056]
  MoveL 1212 to (15.2, -212.53, 388.5) mm, rotated rx -20.64 ry -2.52 rz 0.95 deg; joints [3.212, -139.548, -54.11, -67.056, 93.032, -2.099]
  MoveL 1213 to (15.2, -204.92, 385.16) mm, rotated rx -21.05 ry -2.39 rz 0.92 deg; joints [3.248, -138.534, -55.963, -66.617, 92.877, -2.065]
  MoveL 1214 to (14.78, -195.93, 381.15) mm, rotated rx -22.22 ry -1.94 rz 0.79 deg; joints [3.448, -137.776, -57.071, -67.426, 92.342, -1.872]
  MoveL 1215 to (14.83, -190.5, 379) mm, rotated rx -23.04 ry -1.61 rz 0.69 deg; joints [3.573, -137.434, -57.534, -68.113, 91.958, -1.751]
  MoveL 1216 to (14.75, -184.53, 376.92) mm, rotated rx -22.73 ry -1.18 rz 0.49 deg; joints [3.746, -136.273, -59.928, -66.554, 91.472, -1.578]
  MoveL 1217 to (14.96, -174.73, 372.98) mm, rotated rx -21.38 ry -0.69 rz 0.27 deg; joints [3.91, -133.929, -64.867, -62.592, 90.943, -1.411]
  MoveL 1218 to (14.13, -168.15, 370) mm, rotated rx -20.9 ry -0.61 rz 0.23 deg; joints [3.991, -132.663, -67.421, -60.82, 90.854, -1.329]
  MoveL 1219 to (15.27, -163.69, 368.17) mm, rotated rx -20.89 ry -0.8 rz 0.3 deg; joints [3.812, -132.094, -68.538, -60.271, 91.085, -1.506]
  MoveL 1220 to (14.95, -155.11, 365.36) mm, rotated rx -20.68 ry -1.16 rz 0.44 deg; joints [3.654, -130.94, -70.958, -58.804, 91.508, -1.66]
  MoveL 1221 to (15.12, -145.16, 362.25) mm, rotated rx -20.59 ry -1.05 rz 0.39 deg; joints [3.669, -129.686, -73.556, -57.373, 91.382, -1.646]
  MoveL 1222 to (8.91, -139.55, 360) mm, rotated rx -20.47 ry -1.15 rz 0.43 deg; joints [4.105, -128.786, -75.316, -56.385, 91.419, -1.215]
  MoveL 1223 to (15.82, -139.02, 360.27) mm, rotated rx -20.5 ry -1 rz 0.37 deg; joints [3.619, -128.922, -75.144, -56.456, 91.342, -1.695]
  MoveL 1224 to (14.61, -133.68, 357.94) mm, rotated rx -20.43 ry -0.96 rz 0.36 deg; joints [3.718, -128.164, -76.596, -55.69, 91.288, -1.596]
  MoveL 1225 to (15.28, -124.58, 354.85) mm, rotated rx -20.29 ry -0.91 rz 0.34 deg; joints [3.663, -127.048, -78.887, -54.374, 91.248, -1.649]
  MoveL 1226 to (15.12, -115.92, 351.11) mm, rotated rx -19.67 ry -0.92 rz 0.33 deg; joints [3.647, -125.697, -81.643, -52.351, 91.268, -1.663]
  MoveL 1227 to (9.55, -111.57, 349) mm, rotated rx -19.41 ry -1.07 rz 0.38 deg; joints [4.025, -124.926, -83.132, -51.366, 91.372, -1.29]
  MoveL 1228 to (14.57, -111.57, 349) mm, rotated rx -19.42 ry -0.89 rz 0.31 deg; joints [3.689, -125.019, -82.964, -51.458, 91.24, -1.62]
  MoveL 1229 to (14.92, -105.4, 346.69) mm, rotated rx -19.46 ry -0.88 rz 0.31 deg; joints [3.65, -124.337, -84.288, -50.851, 91.233, -1.659]
  MoveL 1230 to (14.83, -95.74, 344.53) mm, rotated rx -19.55 ry -0.88 rz 0.31 deg; joints [3.637, -123.458, -86.228, -49.885, 91.228, -1.672]
  MoveL 1231 to (14.82, -86.78, 341.4) mm, rotated rx -19.69 ry -0.79 rz 0.28 deg; joints [3.655, -122.539, -88.015, -49.15, 91.136, -1.654]
  MoveL 1232 to (15.04, -81.79, 339) mm, rotated rx -19.94 ry -0.68 rz 0.25 deg; joints [3.682, -122.021, -88.84, -49.095, 91.001, -1.629]
  MoveL 1233 to (14.9, -74.93, 336) mm, rotated rx -20.5 ry -0.47 rz 0.18 deg; joints [3.786, -121.413, -89.757, -49.332, 90.747, -1.529]
  MoveL 1234 to (15.09, -64.65, 332.54) mm, rotated rx -20.73 ry -0.46 rz 0.18 deg; joints [3.748, -120.444, -91.628, -48.663, 90.742, -1.567]
  MoveL 1235 to (15.37, -56.92, 330.54) mm, rotated rx -20.59 ry -0.5 rz 0.19 deg; joints [3.681, -119.687, -93.302, -47.609, 90.799, -1.633]
  MoveL 1236 to (14.45, -52.52, 328.94) mm, rotated rx -20.47 ry -0.59 rz 0.22 deg; joints [3.707, -119.177, -94.33, -46.978, 90.891, -1.607]
  MoveL 1237 to (15.12, -45.36, 326.23) mm, rotated rx -20.05 ry -0.64 rz 0.23 deg; joints [3.597, -118.294, -96.169, -45.603, 90.968, -1.714]
  MoveL 1238 to (14.88, -35.12, 321.59) mm, rotated rx -20.07 ry -0.6 rz 0.22 deg; joints [3.604, -117.136, -98.229, -44.715, 90.933, -1.707]
  MoveL 1239 to (14.92, -24.34, 317.62) mm, rotated rx -19.25 ry -0.76 rz 0.27 deg; joints [3.47, -115.801, -101.094, -42.376, 91.147, -1.834]
  MoveL 1240 to (14.77, -14.25, 314.57) mm, rotated rx -18.71 ry -0.61 rz 0.21 deg; joints [3.526, -114.696, -103.543, -40.489, 90.992, -1.776]
  MoveL 1241 to (15.04, -4.34, 311.63) mm, rotated rx -18.96 ry -0.44 rz 0.15 deg; joints [3.567, -113.878, -105.157, -39.936, 90.797, -1.737]
  MoveL 1242 to (14.98, 5.28, 307.58) mm, rotated rx -19.01 ry -0.49 rz 0.17 deg; joints [3.512, -112.898, -106.905, -39.216, 90.862, -1.791]
  MoveL 1243 to (15.1, 14.86, 304.51) mm, rotated rx -18.79 ry -0.61 rz 0.21 deg; joints [3.396, -111.997, -108.81, -38.002, 91.011, -1.904]
  MoveL 1244 to (15.09, 25.01, 300.85) mm, rotated rx -18.41 ry -0.79 rz 0.26 deg; joints [3.245, -110.964, -110.96, -36.507, 91.243, -2.05]
  MoveL 1245 to (15.1, 35.58, 297.67) mm, rotated rx -18.2 ry -0.72 rz 0.24 deg; joints [3.237, -110.008, -113.018, -35.197, 91.182, -2.056]
  MoveL 1246 to (14.98, 45.13, 294.32) mm, rotated rx -18.2 ry -0.6 rz 0.2 deg; joints [3.288, -109.121, -114.723, -34.375, 91.039, -2.005]
  MoveL 1247 to (14.83, 54.59, 291.44) mm, rotated rx -18.2 ry -0.52 rz 0.17 deg; joints [3.315, -108.317, -116.374, -33.524, 90.952, -1.98]
  MoveL 1248 to (14.84, 64.78, 288.01) mm, rotated rx -17.96 ry -0.61 rz 0.2 deg; joints [3.205, -107.39, -118.311, -32.284, 91.081, -2.085]
  MoveL 1249 to (14.92, 73.34, 285.27) mm, rotated rx -17.53 ry -0.69 rz 0.22 deg; joints [3.099, -106.596, -120.117, -30.847, 91.195, -2.185]
  MoveL 1250 to (25.35, -245.18, 401.78) mm, rotated rx -21 ry -2.56 rz 0.98 deg; joints [2.595, -146.263, -40.643, -74.202, 93.155, -2.711]
  MoveL 1251 to (21.35, -240.18, 399) mm, rotated rx -20.83 ry -2.53 rz 0.96 deg; joints [2.862, -144.826, -43.456, -72.637, 93.087, -2.446]
  MoveL 1252 to (25.01, -234.52, 396.71) mm, rotated rx -20.6 ry -2.61 rz 0.98 deg; joints [2.553, -143.66, -45.863, -71.192, 93.233, -2.75]
  MoveL 1253 to (24.84, -224.87, 392.31) mm, rotated rx -20.35 ry -3.02 rz 1.12 deg; joints [2.364, -141.686, -49.822, -68.979, 93.705, -2.936]
  MoveL 1254 to (24.95, -217.46, 390.06) mm, rotated rx -20.54 ry -2.91 rz 1.09 deg; joints [2.376, -140.603, -52.028, -68.039, 93.579, -2.926]
  MoveL 1255 to (25.38, -212.7, 388.8) mm, rotated rx -20.77 ry -2.84 rz 1.08 deg; joints [2.357, -140.041, -53.175, -67.684, 93.503, -2.946]
  MoveL 1256 to (24.72, -194.78, 382.06) mm, rotated rx -22.94 ry -2.03 rz 0.86 deg; joints [2.693, -138.534, -55.632, -68.86, 92.523, -2.625]
  MoveL 1257 to (20.28, -190.5, 379) mm, rotated rx -23.3 ry -1.62 rz 0.7 deg; joints [3.175, -137.759, -56.849, -68.746, 92.007, -2.147]
  MoveL 1258 to (24.73, -184.65, 377.26) mm, rotated rx -23.16 ry -1.87 rz 0.8 deg; joints [2.726, -136.976, -58.542, -67.721, 92.335, -2.594]
  MoveL 1259 to (25.2, -174.93, 373.1) mm, rotated rx -21.77 ry -1.59 rz 0.63 deg; joints [2.76, -134.58, -63.557, -63.701, 92.067, -2.552]
  MoveL 1260 to (24.61, -163.53, 368.46) mm, rotated rx -20.61 ry -1.4 rz 0.53 deg; joints [2.829, -132.271, -68.381, -60.016, 91.893, -2.475]
  MoveL 1261 to (24.82, -155.08, 365.54) mm, rotated rx -20.58 ry -1.53 rz 0.57 deg; joints [2.725, -131.196, -70.569, -58.879, 92.05, -2.577]
  MoveL 1262 to (24.96, -145.16, 362.42) mm, rotated rx -20.71 ry -1.47 rz 0.55 deg; joints [2.707, -130.056, -72.883, -57.829, 91.983, -2.597]
  MoveL 1263 to (24.94, -138.8, 360.5) mm, rotated rx -20.54 ry -1.39 rz 0.52 deg; joints [2.717, -129.22, -74.654, -56.726, 91.906, -2.585]
  MoveL 1264 to (24.77, -133.15, 357.97) mm, rotated rx -20.63 ry -1.29 rz 0.48 deg; joints [2.757, -128.506, -75.964, -56.218, 91.783, -2.546]
  MoveL 1265 to (25.06, -124.32, 354.23) mm, rotated rx -20.37 ry -1.11 rz 0.41 deg; joints [2.775, -127.253, -78.428, -54.741, 91.603, -2.527]
  MoveL 1266 to (25.34, -115.02, 351.47) mm, rotated rx -19.82 ry -0.93 rz 0.34 deg; joints [2.791, -125.978, -81.216, -52.669, 91.431, -2.506]
  MoveL 1267 to (24.99, -105.28, 347.16) mm, rotated rx -19.31 ry -0.86 rz 0.3 deg; joints [2.806, -124.552, -84.059, -50.731, 91.372, -2.487]
  MoveL 1268 to (24.61, -95.69, 344.85) mm, rotated rx -19.62 ry -0.91 rz 0.33 deg; joints [2.782, -123.751, -85.749, -50.158, 91.422, -2.513]
  MoveL 1269 to (25.16, -86.71, 341.62) mm, rotated rx -20.01 ry -0.61 rz 0.22 deg; joints [2.855, -122.903, -87.298, -49.832, 91.069, -2.445]
  MoveL 1270 to (24.83, -74.5, 336.42) mm, rotated rx -20.59 ry -0.21 rz 0.08 deg; joints [3.043, -121.666, -89.394, -49.533, 90.588, -2.262]
  MoveL 1271 to (25.01, -64.5, 332.52) mm, rotated rx -20.61 ry -0.27 rz 0.1 deg; joints [2.959, -120.593, -91.438, -48.592, 90.665, -2.346]
  MoveL 1272 to (23.44, -57.18, 330.29) mm, rotated rx -20.52 ry -0.38 rz 0.14 deg; joints [3.012, -119.819, -93.049, -47.669, 90.784, -2.293]
  MoveL 1273 to (24.91, -45.6, 326.36) mm, rotated rx -20.16 ry -0.36 rz 0.13 deg; joints [2.836, -118.558, -95.687, -45.932, 90.803, -2.464]
  MoveL 1274 to (25.44, -35.1, 321.88) mm, rotated rx -19.95 ry -0.43 rz 0.15 deg; joints [2.701, -117.358, -97.968, -44.642, 90.904, -2.595]
  MoveL 1275 to (21.65, -30.28, 319) mm, rotated rx -19.57 ry -0.54 rz 0.19 deg; joints [2.969, -116.528, -99.461, -43.597, 90.992, -2.329]
  MoveL 1276 to (17.48, -30.28, 319) mm, rotated rx -19.68 ry -0.59 rz 0.21 deg; joints [3.343, -116.471, -99.503, -43.718, 90.971, -1.961]
  MoveL 1277 to (24.68, -24.1, 317.6) mm, rotated rx -19.09 ry -0.57 rz 0.2 deg; joints [2.627, -115.944, -100.955, -42.219, 91.102, -2.661]
  MoveL 1278 to (24.82, -14.13, 314.15) mm, rotated rx -18.88 ry -0.59 rz 0.2 deg; joints [2.549, -114.928, -103.034, -40.945, 91.15, -2.736]
  MoveL 1279 to (25.19, -4.33, 311.26) mm, rotated rx -19.02 ry -0.63 rz 0.22 deg; joints [2.445, -114.123, -104.68, -40.248, 91.203, -2.839]
  MoveL 1280 to (24.95, 5.38, 308.25) mm, rotated rx -18.9 ry -0.54 rz 0.18 deg; joints [2.467, -113.207, -106.594, -39.128, 91.11, -2.817]
  MoveL 1281 to (25.18, 14.89, 304.67) mm, rotated rx -18.52 ry -0.78 rz 0.26 deg; joints [2.237, -112.226, -108.619, -37.724, 91.434, -3.038]
  MoveL 1282 to (24.92, 24.81, 301.02) mm, rotated rx -18.29 ry -1.14 rz 0.38 deg; joints [1.988, -111.277, -110.544, -36.544, 91.867, -3.28]
  MoveL 1283 to (23.22, 31.12, 300) mm, rotated rx -18.32 ry -1.05 rz 0.35 deg; joints [2.185, -110.813, -111.685, -35.884, 91.737, -3.087]
  MoveL 1284 to (19.97, 31.12, 300) mm, rotated rx -18.24 ry -0.94 rz 0.31 deg; joints [2.598, -110.689, -111.919, -35.676, 91.543, -2.682]
  MoveL 1285 to (25.28, 36.05, 297.67) mm, rotated rx -18.48 ry -0.86 rz 0.29 deg; joints [2.052, -110.349, -112.391, -35.795, 91.551, -3.22]
  MoveL 1286 to (25, 45.17, 294.56) mm, rotated rx -18.45 ry -0.67 rz 0.22 deg; joints [2.14, -109.495, -114.069, -34.929, 91.333, -3.133]
  MoveL 1287 to (24.8, 54.66, 291.54) mm, rotated rx -18.26 ry -0.53 rz 0.17 deg; joints [2.182, -108.618, -115.915, -33.763, 91.19, -3.089]
  MoveL 1288 to (24.99, 60.4, 290) mm, rotated rx -18.03 ry -0.45 rz 0.15 deg; joints [2.166, -108.119, -117.095, -32.853, 91.124, -3.102]
  MoveL 1289 to (17.79, 60.4, 290) mm, rotated rx -18.1 ry -0.49 rz 0.16 deg; joints [2.971, -107.937, -117.332, -32.849, 90.99, -2.315]
  MoveL 1290 to (25.19, 65.24, 288) mm, rotated rx -17.74 ry -0.41 rz 0.13 deg; joints [2.13, -107.583, -118.191, -32.001, 91.097, -3.134]
  MoveL 1291 to (24.78, 73.1, 285.09) mm, rotated rx -17.49 ry -0.36 rz 0.11 deg; joints [2.147, -106.8, -119.778, -30.945, 91.057, -3.115]
  MoveL 1292 to (33.01, -261.48, 407.83) mm, rotated rx -17.37 ry -2.69 rz 0.84 deg; joints [2.035, -146.611, -40.933, -69.976, 93.528, -3.228]
  MoveL 1293 to (25.61, -254.17, 405) mm, rotated rx -19.19 ry -2.74 rz 0.95 deg; joints [2.518, -146.473, -40.667, -72.17, 93.419, -2.773]
  MoveL 1294 to (30.98, -212.81, 389) mm, rotated rx -20.9 ry -3.16 rz 1.21 deg; joints [1.829, -140.403, -52.48, -68.194, 93.926, -3.471]
  MoveL 1295 to (25.57, -205.42, 387.43) mm, rotated rx -21.25 ry -2.65 rz 1.03 deg; joints [2.399, -139.326, -54.685, -67.358, 93.282, -2.908]
  MoveL 1296 to (25.72, -167.84, 370) mm, rotated rx -20.89 ry -1.5 rz 0.57 deg; joints [2.721, -133.039, -66.778, -61.14, 92.006, -2.584]
  MoveL 1297 to (32.82, -161.47, 369) mm, rotated rx -20.66 ry -2.21 rz 0.83 deg; joints [1.842, -132.511, -68.176, -60.108, 92.917, -3.452]
  MoveL 1298 to (25.5, -81.02, 339) mm, rotated rx -20.35 ry -0.34 rz 0.13 deg; joints [2.938, -122.329, -88.216, -49.813, 90.757, -2.364]
  MoveL 1299 to (26.26, -53.82, 328.78) mm, rotated rx -20.41 ry -0.34 rz 0.13 deg; joints [2.762, -119.456, -93.76, -47.21, 90.782, -2.538]
  MoveL 1300 to (28.41, -28.7, 320) mm, rotated rx -19.41 ry -0.53 rz 0.19 deg; joints [2.321, -116.683, -99.58, -43.18, 91.107, -2.965]
  MoveL 1301 to (32.52, 31.12, 300) mm, rotated rx -18.58 ry -0.96 rz 0.32 deg; joints [1.256, -111.124, -111.065, -36.476, 91.805, -4.002]
  MoveL 1302 to (35.06, -254.98, 405.62) mm, rotated rx -19.24 ry -2.63 rz 0.92 deg; joints [1.919, -147.062, -39.532, -72.792, 93.411, -3.363]
  MoveL 1303 to (35.4, -245.33, 402.79) mm, rotated rx -21.02 ry -2.78 rz 1.07 deg; joints [1.825, -146.86, -39.611, -74.709, 93.511, -3.474]
  MoveL 1304 to (35.71, -238.63, 400.54) mm, rotated rx -20.68 ry -3.09 rz 1.17 deg; joints [1.648, -145.265, -42.99, -72.608, 93.886, -3.648]
  MoveL 1305 to (34.7, -232.83, 397.54) mm, rotated rx -20.02 ry -3.04 rz 1.11 deg; joints [1.699, -143.454, -46.7, -70.053, 93.848, -3.59]
  MoveL 1306 to (35.1, -224.44, 393.58) mm, rotated rx -20.28 ry -3.2 rz 1.18 deg; joints [1.57, -142.096, -49.271, -69.111, 94.029, -3.721]
  MoveL 1307 to (35.06, -214.83, 390.66) mm, rotated rx -20.81 ry -3.08 rz 1.17 deg; joints [1.583, -140.899, -51.644, -68.459, 93.88, -3.714]
  MoveL 1308 to (42.27, -208.26, 390) mm, rotated rx -21.51 ry -1.63 rz 0.64 deg; joints [1.639, -140.494, -52.513, -68.617, 92.287, -3.659]
  MoveL 1309 to (35.25, -208.03, 390) mm, rotated rx -21.25 ry -2.88 rz 1.12 deg; joints [1.63, -140.276, -53.059, -68.096, 93.636, -3.671]
  MoveL 1310 to (35.38, -202.95, 387.93) mm, rotated rx -21.86 ry -2.62 rz 1.05 deg; joints [1.71, -139.823, -53.784, -68.416, 93.322, -3.596]
  MoveL 1311 to (34.96, -194.3, 382.57) mm, rotated rx -22.96 ry -2.55 rz 1.08 deg; joints [1.741, -138.944, -54.976, -69.193, 93.193, -3.573]
  MoveL 1312 to (34.89, -184.81, 377.63) mm, rotated rx -23.27 ry -2.8 rz 1.2 deg; joints [1.596, -137.562, -57.483, -68.398, 93.473, -3.721]
  MoveL 1313 to (35.11, -175.04, 373.48) mm, rotated rx -22.16 ry -2.92 rz 1.19 deg; joints [1.457, -135.362, -62.069, -64.916, 93.673, -3.85]
  MoveL 1314 to (35.49, -165.85, 370.69) mm, rotated rx -21.01 ry -2.7 rz 1.04 deg; joints [1.458, -133.452, -66.254, -61.485, 93.481, -3.838]
  MoveL 1315 to (34.78, -154.89, 366.87) mm, rotated rx -20.74 ry -2.08 rz 0.79 deg; joints [1.715, -131.759, -69.705, -59.405, 92.799, -3.578]
  MoveL 1316 to (35.09, -145.51, 363.12) mm, rotated rx -20.82 ry -1.76 rz 0.67 deg; joints [1.787, -130.532, -72.065, -58.339, 92.435, -3.506]
  MoveL 1317 to (35.08, -138.75, 360.48) mm, rotated rx -20.83 ry -1.55 rz 0.59 deg; joints [1.845, -129.643, -73.795, -57.493, 92.207, -3.449]
  MoveL 1318 to (34.97, -132.84, 357.12) mm, rotated rx -20.67 ry -1.44 rz 0.54 deg; joints [1.866, -128.685, -75.54, -56.532, 92.095, -3.426]
  MoveL 1319 to (34.82, -124.31, 353.81) mm, rotated rx -20.57 ry -1.48 rz 0.56 deg; joints [1.814, -127.6, -77.686, -55.384, 92.149, -3.477]
  MoveL 1320 to (35.26, -114.17, 351.57) mm, rotated rx -20.02 ry -1.36 rz 0.5 deg; joints [1.772, -126.327, -80.613, -53.175, 92.056, -3.513]
  MoveL 1321 to (34.77, -104.57, 347.61) mm, rotated rx -19.37 ry -1.1 rz 0.39 deg; joints [1.868, -124.86, -83.624, -50.963, 91.794, -3.41]
  MoveL 1322 to (35.07, -95.5, 344.48) mm, rotated rx -19.73 ry -0.76 rz 0.27 deg; joints [1.966, -123.979, -85.275, -50.525, 91.397, -3.317]
  MoveL 1323 to (35.08, -85.91, 341.02) mm, rotated rx -20.38 ry -0.74 rz 0.27 deg; joints [1.941, -123.195, -86.622, -50.615, 91.342, -3.349]
  MoveL 1324 to (34.97, -80.02, 339) mm, rotated rx -20.72 ry -0.6 rz 0.23 deg; joints [1.993, -122.685, -87.542, -50.534, 91.172, -3.3]
  MoveL 1325 to (34.94, -74.15, 336.88) mm, rotated rx -20.78 ry -0.42 rz 0.16 deg; joints [2.054, -122.053, -88.759, -49.998, 90.971, -3.241]
  MoveL 1326 to (34.96, -64.63, 332.25) mm, rotated rx -20.54 ry -0.27 rz 0.1 deg; joints [2.069, -120.789, -91.09, -48.684, 90.818, -3.223]
  MoveL 1327 to (37.8, -58.66, 330.17) mm, rotated rx -20.54 ry -0.35 rz 0.13 deg; joints [1.74, -120.257, -92.172, -48.138, 90.961, -3.548]
  MoveL 1328 to (34.71, -54.75, 328.42) mm, rotated rx -20.4 ry -0.22 rz 0.08 deg; joints [2.058, -119.661, -93.292, -47.465, 90.777, -3.232]
  MoveL 1329 to (34.85, -45.36, 325.47) mm, rotated rx -20.2 ry -0.33 rz 0.12 deg; joints [1.933, -118.698, -95.322, -46.211, 90.924, -3.354]
  MoveL 1330 to (35.21, -34.67, 321.61) mm, rotated rx -19.61 ry -0.53 rz 0.19 deg; joints [1.717, -117.452, -97.959, -44.246, 91.201, -3.561]
  MoveL 1331 to (35.89, -28.14, 320) mm, rotated rx -19.37 ry -0.65 rz 0.23 deg; joints [1.539, -116.851, -99.375, -43.196, 91.38, -3.733]
  MoveL 1332 to (34.6, -23.15, 317.78) mm, rotated rx -19.15 ry -0.62 rz 0.22 deg; joints [1.637, -116.2, -100.627, -42.372, 91.347, -3.635]
  MoveL 1333 to (34.95, -14.25, 314.81) mm, rotated rx -18.8 ry -0.64 rz 0.22 deg; joints [1.527, -115.268, -102.623, -40.963, 91.402, -3.738]
  MoveL 1334 to (34.83, -4.77, 311.48) mm, rotated rx -19.12 ry -0.62 rz 0.22 deg; joints [1.492, -114.459, -104.09, -40.625, 91.373, -3.776]
  MoveL 1335 to (36.15, -0.26, 309) mm, rotated rx -19.02 ry -0.75 rz 0.26 deg; joints [1.251, -113.943, -104.967, -40.177, 91.558, -4.012]
  MoveL 1336 to (34.96, 5.37, 307.68) mm, rotated rx -18.71 ry -0.73 rz 0.25 deg; joints [1.328, -113.378, -106.315, -39.087, 91.548, -3.932]
  MoveL 1337 to (35.03, 14.88, 304.82) mm, rotated rx -18.22 ry -0.82 rz 0.27 deg; joints [1.18, -112.444, -108.45, -37.409, 91.705, -4.07]
  MoveL 1338 to (35.05, 24.96, 301.52) mm, rotated rx -18.25 ry -0.93 rz 0.31 deg; joints [1.037, -111.58, -110.189, -36.575, 91.844, -4.211]
  MoveL 1339 to (35.14, 35.8, 297.59) mm, rotated rx -18.72 ry -0.89 rz 0.3 deg; joints [0.978, -110.698, -111.685, -36.431, 91.781, -4.276]
  MoveL 1340 to (35.06, 45.24, 295.01) mm, rotated rx -18.55 ry -0.83 rz 0.28 deg; joints [0.94, -109.894, -113.491, -35.247, 91.733, -4.311]
  MoveL 1341 to (34.84, 54.68, 291.72) mm, rotated rx -18.39 ry -0.62 rz 0.21 deg; joints [1.001, -108.981, -115.325, -34.156, 91.517, -4.248]
  MoveL 1342 to (35.22, 60.4, 290) mm, rotated rx -18.07 ry -0.65 rz 0.21 deg; joints [0.877, -108.461, -116.556, -33.128, 91.594, -4.365]
  MoveL 1343 to (34.96, 65.21, 287.88) mm, rotated rx -17.81 ry -0.68 rz 0.22 deg; joints [0.829, -107.918, -117.622, -32.352, 91.654, -4.408]
  MoveL 1344 to (35.31, 74.15, 285.05) mm, rotated rx -17.24 ry -0.77 rz 0.24 deg; joints [0.618, -107.098, -119.582, -30.652, 91.838, -4.605]
  MoveL 1345 to (37.65, 81.64, 284.5) mm, rotated rx -17.01 ry -0.84 rz 0.26 deg; joints [0.217, -106.816, -120.827, -29.482, 92.012, -4.991]
  MoveL 1346 to (44.97, -254.26, 403.39) mm, rotated rx -19.49 ry -2.61 rz 0.92 deg; joints [1.249, -147.311, -38.716, -73.655, 93.495, -4.026]
  MoveL 1347 to (44.75, -245.49, 402.86) mm, rotated rx -20.15 ry -2.87 rz 1.05 deg; joints [1.135, -146.465, -40.671, -73.229, 93.765, -4.148]
  MoveL 1348 to (44.34, -238.18, 400.59) mm, rotated rx -20.35 ry -3.16 rz 1.17 deg; joints [1.019, -145.264, -43.141, -72.183, 94.074, -4.266]
  MoveL 1349 to (45.41, -232.8, 398.05) mm, rotated rx -20.32 ry -2.96 rz 1.1 deg; joints [0.991, -144.134, -45.359, -71.055, 93.87, -4.293]
  MoveL 1350 to (45.09, -223.93, 394.45) mm, rotated rx -20.84 ry -2.18 rz 0.83 deg; joints [1.283, -142.718, -48.014, -70.266, 92.963, -4.007]
  MoveL 1351 to (45.01, -214.27, 391.67) mm, rotated rx -21.23 ry -1.35 rz 0.53 deg; joints [1.578, -141.267, -50.94, -69.117, 92.015, -3.716]
  MoveL 1352 to (45.44, -203.82, 387.5) mm, rotated rx -21.92 ry -1.01 rz 0.41 deg; joints [1.649, -139.951, -53.38, -68.657, 91.601, -3.652]
  MoveL 1353 to (44.9, -195, 383.03) mm, rotated rx -22.54 ry -1.49 rz 0.62 deg; joints [1.456, -138.909, -55.169, -68.567, 92.111, -3.849]
  MoveL 1354 to (46.37, -188.56, 380.42) mm, rotated rx -22.7 ry -1.73 rz 0.72 deg; joints [1.222, -138.077, -56.789, -67.964, 92.384, -4.084]
  MoveL 1355 to (44.68, -184.07, 378.15) mm, rotated rx -22.72 ry -2.31 rz 0.97 deg; joints [1.078, -137.387, -58.095, -67.411, 93.025, -4.229]
  MoveL 1356 to (45, -175.51, 374.48) mm, rotated rx -21.96 ry -2.9 rz 1.17 deg; joints [0.734, -135.702, -61.607, -64.888, 93.758, -4.566]
  MoveL 1357 to (44.46, -165.4, 371.28) mm, rotated rx -21.36 ry -3.15 rz 1.23 deg; joints [0.59, -134.018, -65.227, -62.374, 94.082, -4.703]
  MoveL 1358 to (48.19, -160.4, 369) mm, rotated rx -21.41 ry -2.95 rz 1.16 deg; joints [0.363, -133.402, -66.384, -61.885, 93.892, -4.928]
  MoveL 1359 to (45, -154.56, 366.58) mm, rotated rx -21.34 ry -2.72 rz 1.06 deg; joints [0.665, -132.423, -68.281, -60.869, 93.602, -4.627]
  MoveL 1360 to (45.08, -145.43, 363.36) mm, rotated rx -21.42 ry -2.2 rz 0.86 deg; joints [0.827, -131.214, -70.667, -59.719, 93.023, -4.465]
  MoveL 1361 to (45.22, -138.44, 360.52) mm, rotated rx -21.12 ry -1.9 rz 0.73 deg; joints [0.896, -130.105, -72.897, -58.278, 92.71, -4.392]
  MoveL 1362 to (44.51, -132.9, 357.85) mm, rotated rx -20.74 ry -1.7 rz 0.64 deg; joints [0.994, -129.11, -74.86, -56.91, 92.506, -4.289]
  MoveL 1363 to (44.95, -124.54, 354.75) mm, rotated rx -20.57 ry -1.72 rz 0.65 deg; joints [0.892, -128.034, -77.042, -55.639, 92.554, -4.389]
  MoveL 1364 to (45.11, -114.01, 350.98) mm, rotated rx -20.04 ry -1.81 rz 0.66 deg; joints [0.754, -126.591, -80.076, -53.532, 92.702, -4.518]
  MoveL 1365 to (45.25, -108.23, 350) mm, rotated rx -19.89 ry -1.68 rz 0.61 deg; joints [0.76, -125.979, -81.524, -52.538, 92.575, -4.509]
  MoveL 1366 to (44.99, -104.35, 347.92) mm, rotated rx -19.99 ry -1.43 rz 0.52 deg; joints [0.872, -125.464, -82.385, -52.275, 92.287, -4.4]
  MoveL 1367 to (44.86, -95.71, 344.17) mm, rotated rx -20.08 ry -0.87 rz 0.32 deg; joints [1.094, -124.376, -84.385, -51.395, 91.642, -4.181]
  MoveL 1368 to (44.78, -86.05, 341.02) mm, rotated rx -20.4 ry -0.71 rz 0.26 deg; joints [1.124, -123.467, -86.139, -50.865, 91.447, -4.154]
  MoveL 1369 to (44.54, -80.55, 339) mm, rotated rx -20.79 ry -0.74 rz 0.28 deg; joints [1.103, -123.024, -86.89, -50.948, 91.461, -4.18]
  MoveL 1370 to (45.28, -74.75, 336.89) mm, rotated rx -20.88 ry -0.84 rz 0.32 deg; joints [0.953, -122.468, -87.968, -50.521, 91.587, -4.33]
  MoveL 1371 to (45, -64.62, 333.12) mm, rotated rx -20.56 ry -0.87 rz 0.33 deg; joints [0.883, -121.255, -90.43, -48.964, 91.645, -4.394]
  MoveL 1372 to (45.16, -57.41, 330.62) mm, rotated rx -20.6 ry -0.85 rz 0.32 deg; joints [0.828, -120.529, -91.863, -48.292, 91.631, -4.45]
  MoveL 1373 to (44.87, -52.76, 328.52) mm, rotated rx -20.3 ry -0.76 rz 0.28 deg; joints [0.853, -119.866, -93.176, -47.334, 91.554, -4.421]
  MoveL 1374 to (45.06, -45.36, 325.46) mm, rotated rx -20.01 ry -0.91 rz 0.33 deg; joints [0.692, -118.989, -94.919, -46.2, 91.76, -4.576]
  MoveL 1375 to (45.07, -34.68, 321.5) mm, rotated rx -19.41 ry -1.33 rz 0.47 deg; joints [0.362, -117.765, -97.514, -44.277, 92.308, -4.893]
  MoveL 1376 to (45.14, -27.86, 320) mm, rotated rx -19.35 ry -1.48 rz 0.52 deg; joints [0.218, -117.216, -98.808, -43.488, 92.499, -5.034]
  MoveL 1377 to (44.89, -22.72, 318.21) mm, rotated rx -19.07 ry -1.44 rz 0.5 deg; joints [0.209, -116.618, -100.085, -42.528, 92.476, -5.039]
  MoveL 1378 to (45.09, -14.37, 315.31) mm, rotated rx -18.9 ry -1.24 rz 0.43 deg; joints [0.211, -115.746, -101.868, -41.425, 92.288, -5.033]
  MoveL 1379 to (45, -4.72, 311.68) mm, rotated rx -19.12 ry -1.07 rz 0.37 deg; joints [0.237, -114.842, -103.506, -40.903, 92.079, -5.011]
  MoveL 1380 to (45.1, -0.26, 309) mm, rotated rx -18.9 ry -1.1 rz 0.38 deg; joints [0.152, -114.223, -104.572, -40.241, 92.148, -5.091]
  MoveL 1381 to (44.98, 5.37, 307.5) mm, rotated rx -18.73 ry -1.18 rz 0.4 deg; joints [0.063, -113.721, -105.725, -39.432, 92.259, -5.176]
  MoveL 1382 to (45.05, 14.9, 305.24) mm, rotated rx -18.37 ry -1 rz 0.33 deg; joints [0.054, -112.86, -107.789, -37.852, 92.101, -5.178]
  MoveL 1383 to (45.09, 25.09, 302.03) mm, rotated rx -18.25 ry -0.69 rz 0.23 deg; joints [0.122, -111.903, -109.787, -36.658, 91.775, -5.107]
  MoveL 1384 to (46.46, 31.72, 300) mm, rotated rx -18.56 ry -0.8 rz 0.27 deg; joints [-0.137, -111.484, -110.571, -36.621, 91.913, -5.367]
  MoveL 1385 to (44.48, 35.82, 298.29) mm, rotated rx -18.73 ry -0.79 rz 0.27 deg; joints [0.041, -111.06, -111.245, -36.534, 91.859, -5.196]
  MoveL 1386 to (45.04, 44.61, 295.05) mm, rotated rx -18.61 ry -0.68 rz 0.23 deg; joints [-0.048, -110.222, -112.894, -35.601, 91.764, -5.281]
  MoveL 1387 to (45.04, 54.46, 291.25) mm, rotated rx -18.33 ry -0.61 rz 0.2 deg; joints [-0.131, -109.225, -114.877, -34.331, 91.736, -5.357]
  MoveL 1388 to (44.95, 60.4, 290) mm, rotated rx -18.01 ry -0.7 rz 0.23 deg; joints [-0.256, -108.762, -116.131, -33.228, 91.883, -5.473]
  MoveL 1389 to (44.92, 64.98, 288.55) mm, rotated rx -17.69 ry -0.68 rz 0.22 deg; joints [-0.309, -108.314, -117.191, -32.298, 91.9, -5.518]
  MoveL 1390 to (45.14, 75.07, 284.89) mm, rotated rx -17.11 ry -0.73 rz 0.22 deg; joints [-0.526, -107.333, -119.368, -30.538, 92.058, -5.718]
  MoveL 1391 to (45.71, 83.31, 283.38) mm, rotated rx -17.15 ry -0.69 rz 0.21 deg; joints [-0.66, -106.861, -120.64, -29.779, 92.041, -5.849]
  MoveL 1392 to (56.49, -260.52, 408) mm, rotated rx -19.21 ry -2.26 rz 0.79 deg; joints [0.635, -149.178, -35.337, -74.899, 93.26, -4.626]
